C07282=1015.602,-60.319,395.785,165.379,57.389,160.207
C07283=1015.597,-60.568,395.794,165.376,57.396,160.208
C07284=1015.592,-60.819,395.805,165.373,57.403,160.208
C07285=1015.587,-61.068,395.815,165.370,57.410,160.209
C07286=1015.582,-61.318,395.825,165.367,57.417,160.210
C07287=1015.577,-61.568,395.835,165.364,57.424,160.210
C07288=1015.572,-61.818,395.845,165.361,57.431,160.211
C07289=1015.567,-62.067,395.855,165.358,57.438,160.211
C07290=1015.562,-62.317,395.865,165.356,57.444,160.212
C07291=1015.557,-62.567,395.875,165.353,57.451,160.212
C07292=1015.551,-62.817,395.885,165.351,57.458,160.213
C07293=1015.546,-63.066,395.895,165.348,57.465,160.213
C07294=1015.541,-63.316,395.905,165.345,57.472,160.214
C07295=1015.536,-63.566,395.915,165.342,57.479,160.215
C07296=1015.531,-63.816,395.925,165.339,57.486,160.215
C07297=1015.526,-64.065,395.935,165.337,57.493,160.216
C07298=1015.521,-64.315,395.945,165.334,57.500,160.216
C07299=1015.516,-64.565,395.955,165.331,57.507,160.217
C07300=1015.511,-64.814,395.964,165.328,57.514,160.217
C07301=1015.505,-65.064,395.975,165.325,57.521,160.218
C07302=1015.501,-65.314,395.984,165.322,57.528,160.218
C07303=1015.496,-65.563,395.994,165.320,57.534,160.219
C07304=1015.490,-65.813,396.004,165.317,57.541,160.219
C07305=1015.485,-66.063,396.014,165.314,57.548,160.220
C07306=1015.480,-66.313,396.024,165.311,57.555,160.220
C07307=1015.475,-66.562,396.034,165.308,57.562,160.221
C07308=1015.471,-66.812,396.043,165.306,57.568,160.222
C07309=1015.465,-67.062,396.053,165.303,57.575,160.222
C07310=1015.460,-67.312,396.063,165.300,57.582,160.223
C07311=1015.456,-67.561,396.073,165.297,57.589,160.223
C07312=1015.450,-67.811,396.083,165.295,57.595,160.224
C07313=1015.445,-68.061,396.093,165.292,57.602,160.224
C07314=1015.440,-68.310,396.103,165.289,57.609,160.225
C07315=1015.435,-68.561,396.112,165.286,57.616,160.225
C07316=1015.431,-68.811,396.123,165.284,57.622,160.226
C07317=1015.426,-69.060,396.132,165.281,57.629,160.226
C07318=1015.421,-69.323,396.142,165.278,57.636,160.227
C07319=1015.415,-69.600,396.154,165.274,57.644,160.227
C07320=1015.410,-69.877,396.164,165.272,57.651,160.228
C07321=1015.404,-70.154,396.176,165.269,57.659,160.229
C07322=1015.399,-70.432,396.186,165.266,57.667,160.229
C07323=1015.394,-70.682,396.196,165.263,57.673,160.230
C07324=1015.389,-70.931,396.206,165.260,57.680,160.230
C07325=1015.384,-71.182,396.215,165.257,57.687,160.231
C07326=1015.379,-71.431,396.225,165.255,57.692,160.231
C07327=1015.374,-71.681,396.235,165.252,57.700,160.232
C07328=1015.370,-71.930,396.245,165.249,57.707,160.232
C07329=1015.364,-72.181,396.254,165.246,57.713,160.232
C07330=1015.360,-72.430,396.264,165.244,57.719,160.233
C07331=1015.355,-72.680,396.274,165.241,57.726,160.234
C07332=1015.350,-72.930,396.283,165.237,57.733,160.234
C07333=1015.345,-73.180,396.293,165.236,57.739,160.235
C07334=1015.340,-73.429,396.303,165.232,57.746,160.235
C07335=1015.335,-73.678,396.313,165.229,57.753,160.235
C07336=1015.331,-73.928,396.322,165.227,57.759,160.236
C07337=1015.325,-74.179,396.332,165.224,57.766,160.236
C07338=1015.320,-74.428,396.342,165.221,57.773,160.237
C07339=1015.316,-74.678,396.351,165.219,57.779,160.237
C07340=1015.310,-74.927,396.360,165.216,57.786,160.238
C07341=1015.306,-75.177,396.369,165.213,57.793,160.238
C07342=1015.300,-75.427,396.379,165.210,57.800,160.239
C07343=1015.295,-75.677,396.388,165.207,57.806,160.239
C07344=1015.290,-75.926,396.397,165.205,57.813,160.240
C07345=1015.286,-76.176,396.407,165.202,57.820,160.240
C07346=1015.281,-76.426,396.416,165.199,57.827,160.241
C07347=1015.276,-76.676,396.425,165.196,57.833,160.241
C07348=1015.270,-76.926,396.434,165.194,57.840,160.242
C07349=1015.266,-77.176,396.444,165.191,57.847,160.243
C07350=1015.260,-77.425,396.453,165.187,57.853,160.243
C07351=1015.255,-77.675,396.462,165.185,57.860,160.243
C07352=1015.251,-77.925,396.471,165.182,57.867,160.244
C07353=1015.246,-78.175,396.480,165.180,57.874,160.245
C07354=1015.241,-78.424,396.490,165.176,57.880,160.245
C07355=1015.236,-78.675,396.499,165.174,57.887,160.246
C07356=1015.231,-78.924,396.509,165.171,57.893,160.246
C07357=1015.226,-79.174,396.517,165.168,57.900,160.246
C07358=1015.221,-79.424,396.526,165.166,57.907,160.247
C07359=1015.216,-79.673,396.536,165.163,57.913,160.247
C07360=1015.211,-79.923,396.545,165.160,57.920,160.248
C07361=1015.207,-80.173,396.554,165.158,57.927,160.249
///RCONF 1,0,0,0,1,0,0,0,0,0,0,0,0,0,0,0,0,0,0,0,0,0,0,0
C07362=1015.201,-80.423,396.564,165.155,57.933,160.249
C07363=1015.196,-80.673,396.572,165.152,57.940,160.249
C07364=1015.191,-80.923,396.582,165.149,57.947,160.250
C07365=1015.186,-81.173,396.590,165.146,57.954,160.250
C07366=1015.181,-81.423,396.599,165.144,57.960,160.251
C07367=1015.176,-81.672,396.608,165.141,57.967,160.251
C07368=1015.171,-81.921,396.617,165.138,57.974,160.252
C07369=1015.166,-82.171,396.626,165.135,57.981,160.252
C07370=1015.161,-82.421,396.634,165.131,57.988,160.253
C07371=1015.156,-82.671,396.643,165.130,57.994,160.253
C07372=1015.151,-82.921,396.652,165.127,58.001,160.254
C07373=1015.147,-83.171,396.661,165.123,58.008,160.254
C07374=1015.141,-83.421,396.670,165.120,58.015,160.255
C07375=1015.136,-83.670,396.679,165.119,58.021,160.255
C07376=1015.131,-83.920,396.688,165.115,58.028,160.256
C07377=1015.126,-84.169,396.696,165.112,58.035,160.256
C07378=1015.121,-84.419,396.705,165.109,58.042,160.257
C07379=1015.116,-84.669,396.714,165.107,58.048,160.257
C07380=1015.111,-84.919,396.722,165.104,58.055,160.258
C07381=1015.106,-85.169,396.731,165.101,58.062,160.258
C07382=1015.101,-85.419,396.740,165.098,58.068,160.258
C07383=1015.095,-85.698,396.750,165.096,58.076,160.259
C07384=1015.090,-85.978,396.760,165.093,58.083,160.260
C07385=1015.085,-86.257,396.769,165.089,58.090,160.260
C07386=1015.079,-86.536,396.779,165.086,58.098,160.261
C07387=1015.074,-86.786,396.788,165.083,58.105,160.261
C07388=1015.069,-87.036,396.797,165.081,58.111,160.262
C07389=1015.064,-87.285,396.806,165.078,58.118,160.262
C07390=1015.059,-87.535,396.815,165.074,58.124,160.262
C07391=1015.054,-87.785,396.823,165.073,58.131,160.263
C07392=1015.049,-88.035,396.832,165.069,58.137,160.263
C07393=1015.044,-88.285,396.841,165.066,58.144,160.264
C07394=1015.039,-88.535,396.849,165.064,58.150,160.264
C07395=1015.035,-88.784,396.858,165.061,58.157,160.265
C07396=1015.030,-89.034,396.866,165.058,58.163,160.265
C07397=1015.025,-89.283,396.875,165.056,58.170,160.266
C07398=1015.020,-89.534,396.883,165.053,58.176,160.266
C07399=1015.015,-89.784,396.892,165.050,58.183,160.266
C07400=1015.011,-90.034,396.901,165.047,58.189,160.267
C07401=1015.005,-90.284,396.909,165.044,58.196,160.267
C07402=1015.000,-90.533,396.918,165.042,58.202,160.268
C07403=1014.996,-90.783,396.926,165.039,58.209,160.268
C07404=1014.991,-91.032,396.935,165.036,58.216,160.269
C07405=1014.986,-91.282,396.944,165.033,58.222,160.269
C07406=1014.981,-91.532,396.952,165.031,58.229,160.270
C07407=1014.976,-91.782,396.961,165.028,58.235,160.270
C07408=1014.972,-92.032,396.969,165.025,58.241,160.270
C07409=1014.967,-92.281,396.977,165.023,58.248,160.271
C07410=1014.962,-92.531,396.987,165.020,58.254,160.271
C07411=1014.957,-92.781,396.995,165.016,58.260,160.271
C07412=1014.952,-93.031,397.003,165.014,58.267,160.272
C07413=1014.947,-93.281,397.013,165.011,58.273,160.272
C07414=1014.942,-93.531,397.021,165.009,58.279,160.273
C07415=1014.939,-93.781,397.029,165.005,58.286,160.273
C07416=1014.933,-94.030,397.038,165.003,58.292,160.274
C07417=1014.928,-94.280,397.046,165.000,58.299,160.274
C07418=1014.923,-94.530,397.055,164.998,58.305,160.274
C07419=1014.919,-94.779,397.063,164.995,58.312,160.275
C07420=1014.915,-95.030,397.072,164.992,58.318,160.275
C07421=1014.909,-95.279,397.080,164.989,58.324,160.276
C07422=1014.904,-95.529,397.089,164.987,58.330,160.276
C07423=1014.900,-95.778,397.097,164.983,58.336,160.276
C07424=1014.895,-96.029,397.105,164.981,58.343,160.277
C07425=1014.890,-96.278,397.114,164.978,58.349,160.277
C07426=1014.885,-96.528,397.123,164.976,58.355,160.278
C07427=1014.881,-96.777,397.131,164.972,58.362,160.278
C07428=1014.876,-97.028,397.139,164.970,58.368,160.278
C07429=1014.871,-97.278,397.148,164.968,58.374,160.279
C07430=1014.866,-97.528,397.156,164.965,58.381,160.279
C07431=1014.862,-97.777,397.165,164.962,58.387,160.280
C07432=1014.857,-98.027,397.173,164.959,58.393,160.280
C07433=1014.852,-98.277,397.181,164.957,58.399,160.280
C07434=1014.847,-98.527,397.188,164.953,58.405,160.281
C07435=1014.843,-98.777,397.198,164.951,58.412,160.281
C07436=1014.838,-99.027,397.205,164.948,58.418,160.282
C07437=1014.833,-99.276,397.213,164.945,58.425,160.282
C07438=1014.828,-99.526,397.221,164.943,58.431,160.282
C07439=1014.823,-99.776,397.230,164.939,58.438,160.283
C07440=1014.819,-100.026,397.237,164.937,58.444,160.283
C07441=1014.813,-100.275,397.246,164.934,58.450,160.283
C07442=1014.808,-100.526,397.253,164.932,58.457,160.284
C07443=1014.804,-100.775,397.261,164.929,58.463,160.284
C07444=1014.799,-101.025,397.269,164.926,58.469,160.285
C07445=1014.794,-101.275,397.278,164.923,58.475,160.285
C07446=1014.790,-101.525,397.286,164.920,58.481,160.285
C07447=1014.784,-101.806,397.295,164.918,58.488,160.286
C07448=1014.779,-102.088,397.304,164.915,58.496,160.286
C07449=1014.773,-102.369,397.313,164.911,58.503,160.287
C07450=1014.768,-102.651,397.322,164.908,58.510,160.287
C07451=1014.763,-102.900,397.330,164.906,58.516,160.288
C07452=1014.758,-103.150,397.338,164.902,58.523,160.288
C07453=1014.754,-103.399,397.346,164.900,58.529,160.288
C07454=1014.749,-103.650,397.354,164.897,58.535,160.289
C07455=1014.744,-103.900,397.361,164.894,58.541,160.289
C07456=1014.739,-104.149,397.370,164.892,58.547,160.289
C07457=1014.734,-104.399,397.377,164.889,58.554,160.290
C07458=1014.730,-104.649,397.385,164.887,58.560,160.290
C07459=1014.725,-104.899,397.393,164.883,58.566,160.291
C07460=1014.720,-105.148,397.401,164.881,58.572,160.291
C07461=1014.715,-105.399,397.408,164.879,58.578,160.291
C07462=1014.711,-105.648,397.417,164.875,58.585,160.292
C07463=1014.706,-105.898,397.425,164.873,58.590,160.292
C07464=1014.702,-106.148,397.432,164.870,58.597,160.292
C07465=1014.697,-106.398,397.441,164.867,58.603,160.293
C07466=1014.692,-106.648,397.449,164.865,58.609,160.293
C07467=1014.688,-106.898,397.456,164.862,58.615,160.293
C07468=1014.683,-107.148,397.464,164.859,58.621,160.294
C07469=1014.678,-107.397,397.472,164.856,58.627,160.294
C07470=1014.673,-107.647,397.480,164.853,58.633,160.294
C07471=1014.669,-107.897,397.487,164.851,58.639,160.295
C07472=1014.664,-108.147,397.495,164.848,58.646,160.295
C07473=1014.659,-108.396,397.503,164.845,58.652,160.296
C07474=1014.654,-108.646,397.510,164.843,58.658,160.296
C07475=1014.649,-108.896,397.518,164.840,58.664,160.296
C07476=1014.645,-109.146,397.525,164.837,58.670,160.297
C07477=1014.640,-109.396,397.533,164.834,58.676,160.297
C07478=1014.635,-109.646,397.540,164.832,58.682,160.297
C07479=1014.630,-109.896,397.548,164.829,58.688,160.298
C07480=1014.626,-110.145,397.555,164.826,58.695,160.298
C07481=1014.621,-110.395,397.564,164.824,58.701,160.298
C07482=1014.616,-110.645,397.571,164.821,58.707,160.299
C07483=1014.611,-110.894,397.578,164.818,58.713,160.299
C07484=1014.606,-111.144,397.586,164.816,58.719,160.299
C07485=1014.602,-111.394,397.593,164.812,58.725,160.300
C07486=1014.597,-111.644,397.601,164.810,58.731,160.300
C07487=1014.593,-111.894,397.608,164.808,58.737,160.300
C07488=1014.588,-112.144,397.616,164.805,58.743,160.301
C07489=1014.583,-112.394,397.623,164.802,58.750,160.301
C07490=1014.579,-112.644,397.631,164.800,58.756,160.302
C07491=1014.573,-112.894,397.638,164.797,58.762,160.302
C07492=1014.569,-113.143,397.645,164.794,58.768,160.302
C07493=1014.564,-113.393,397.653,164.791,58.774,160.303
C07494=1014.560,-113.643,397.661,164.789,58.779,160.303
C07495=1014.555,-113.893,397.668,164.786,58.785,160.303
C07496=1014.551,-114.143,397.675,164.783,58.792,160.303
C07497=1014.546,-114.393,397.683,164.781,58.798,160.304
C07498=1014.541,-114.643,397.691,164.778,58.804,160.304
C07499=1014.536,-114.892,397.697,164.776,58.810,160.305
C07500=1014.531,-115.142,397.705,164.772,58.815,160.305
C07501=1014.527,-115.392,397.713,164.770,58.821,160.305
C07502=1014.523,-115.641,397.720,164.767,58.827,160.305
C07503=1014.517,-115.891,397.727,164.764,58.834,160.306
C07504=1014.513,-116.141,397.735,164.762,58.840,160.306
C07505=1014.508,-116.391,397.742,164.759,58.845,160.306
C07506=1014.504,-116.642,397.749,164.757,58.851,160.307
C07507=1014.499,-116.891,397.756,164.753,58.857,160.307
C07508=1014.494,-117.141,397.763,164.751,58.863,160.307
C07509=1014.490,-117.390,397.771,164.748,58.869,160.308
C07510=1014.485,-117.641,397.778,164.746,58.875,160.308
C07511=1014.480,-117.922,397.786,164.743,58.881,160.308
C07512=1014.474,-118.204,397.794,164.739,58.888,160.308
C07513=1014.469,-118.485,397.802,164.737,58.895,160.309
C07514=1014.464,-118.767,397.811,164.733,58.901,160.309
C07515=1014.460,-119.017,397.817,164.731,58.907,160.310
C07516=1014.455,-119.266,397.824,164.729,58.913,160.310
C07517=1014.450,-119.517,397.832,164.726,58.919,160.310
C07518=1014.445,-119.766,397.839,164.723,58.925,160.311
C07519=1014.441,-120.016,397.846,164.720,58.931,160.311
C07520=1014.436,-120.266,397.853,164.718,58.937,160.311
C07521=1014.431,-120.516,397.861,164.715,58.942,160.311
C07522=1014.427,-120.766,397.868,164.712,58.948,160.312
C07523=1014.422,-121.016,397.874,164.710,58.954,160.312
C07524=1014.418,-121.265,397.881,164.707,58.959,160.312
C07525=1014.413,-121.515,397.889,164.704,58.966,160.313
C07526=1014.408,-121.766,397.895,164.702,58.972,160.313
C07527=1014.403,-122.015,397.903,164.699,58.977,160.313
C07528=1014.399,-122.265,397.910,164.696,58.983,160.313
C07529=1014.394,-122.515,397.916,164.694,58.989,160.314
C07530=1014.390,-122.764,397.924,164.691,58.994,160.314
C07531=1014.386,-123.014,397.931,164.689,59.000,160.314
C07532=1014.380,-123.265,397.937,164.686,59.006,160.315
C07533=1014.376,-123.514,397.945,164.684,59.012,160.315
C07534=1014.372,-123.765,397.952,164.680,59.018,160.315
C07535=1014.367,-124.014,397.958,164.677,59.023,160.315
C07536=1014.362,-124.264,397.966,164.675,59.029,160.316
C07537=1014.358,-124.514,397.972,164.672,59.034,160.316
C07538=1014.353,-124.763,397.979,164.670,59.040,160.316
C07539=1014.349,-125.013,397.986,164.667,59.046,160.316
C07540=1014.343,-125.263,397.993,164.665,59.052,160.317
C07541=1014.339,-125.514,398.000,164.662,59.058,160.317
C07542=1014.334,-125.763,398.007,164.659,59.063,160.317
C07543=1014.330,-126.013,398.013,164.657,59.069,160.318
C07544=1014.325,-126.263,398.020,164.654,59.074,160.318
C07545=1014.321,-126.513,398.027,164.652,59.080,160.318
C07546=1014.316,-126.762,398.034,164.650,59.086,160.319
C07547=1014.312,-127.012,398.040,164.647,59.091,160.319
C07548=1014.307,-127.262,398.047,164.643,59.098,160.319
C07549=1014.303,-127.512,398.054,164.641,59.103,160.319
C07550=1014.298,-127.761,398.061,164.638,59.109,160.320
C07551=1014.294,-128.012,398.067,164.635,59.114,160.320
C07552=1014.289,-128.261,398.074,164.633,59.120,160.320
C07553=1014.284,-128.511,398.082,164.631,59.125,160.320
C07554=1014.281,-128.760,398.090,164.628,59.130,160.320
C07555=1014.277,-129.009,398.098,164.625,59.134,160.320
C07556=1014.274,-129.259,398.107,164.623,59.136,160.320
C07557=1014.272,-129.509,398.117,164.620,59.140,160.320
C07558=1014.269,-129.759,398.127,164.618,59.143,160.320
C07559=1014.266,-130.008,398.138,164.617,59.144,160.320
C07560=1014.265,-130.258,398.149,164.613,59.146,160.319
C07561=1014.264,-130.507,398.162,164.611,59.146,160.318
C07562=1014.263,-130.757,398.174,164.609,59.147,160.318
C07563=1014.262,-131.006,398.188,164.607,59.147,160.317
C07564=1014.262,-131.256,398.202,164.605,59.146,160.317
C07565=1014.261,-131.506,398.216,164.602,59.145,160.316
C07566=1014.262,-131.755,398.231,164.601,59.143,160.315
C07567=1014.263,-132.005,398.247,164.599,59.141,160.314
C07568=1014.264,-132.255,398.263,164.597,59.138,160.313
C07569=1014.264,-132.505,398.281,164.594,59.135,160.311
C07570=1014.267,-132.754,398.298,164.593,59.132,160.310
C07571=1014.269,-133.004,398.316,164.591,59.128,160.309
C07572=1014.271,-133.254,398.335,164.589,59.122,160.307
C07573=1014.274,-133.504,398.354,164.587,59.117,160.306
C07574=1014.277,-133.753,398.374,164.585,59.111,160.304
C07575=1014.043,-133.779,397.962,164.561,59.455,160.360
C07576=1014.040,-133.530,397.942,164.563,59.460,160.362
C07577=1014.036,-133.281,397.922,164.565,59.466,160.363
C07578=1014.035,-133.031,397.904,164.567,59.470,160.365
C07579=1014.032,-132.780,397.885,164.569,59.474,160.366
C07580=1014.031,-132.531,397.868,164.571,59.478,160.368
C07581=1014.029,-132.282,397.851,164.573,59.482,160.369
C07582=1014.028,-132.032,397.834,164.575,59.484,160.370
C07583=1014.028,-131.782,397.819,164.576,59.486,160.371
C07584=1014.027,-131.533,397.804,164.579,59.488,160.372
C07585=1014.027,-131.283,397.789,164.580,59.489,160.372
C07586=1014.027,-131.033,397.775,164.583,59.490,160.373
C07587=1014.028,-130.783,397.762,164.585,59.490,160.374
C07588=1014.029,-130.534,397.749,164.588,59.490,160.375
C07589=1014.030,-130.284,397.736,164.590,59.489,160.375
C07590=1014.032,-130.035,397.725,164.592,59.487,160.375
C07591=1014.034,-129.785,397.714,164.595,59.485,160.376
C07592=1014.037,-129.535,397.704,164.596,59.483,160.376
C07593=1014.039,-129.285,397.694,164.599,59.480,160.376
C07594=1014.043,-129.036,397.685,164.601,59.477,160.376
C07595=1014.046,-128.786,397.676,164.604,59.473,160.376
C07596=1014.050,-128.536,397.668,164.607,59.469,160.377
C07597=1014.054,-128.287,397.661,164.609,59.464,160.376
C07598=1014.059,-128.037,397.655,164.612,59.459,160.376
C07599=1014.063,-127.788,397.647,164.614,59.453,160.376
C07600=1014.068,-127.539,397.641,164.617,59.447,160.376
C07601=1014.072,-127.288,397.634,164.620,59.442,160.375
C07602=1014.077,-127.038,397.628,164.622,59.436,160.375
C07603=1014.081,-126.789,397.620,164.625,59.431,160.375
C07604=1014.086,-126.539,397.614,164.628,59.425,160.375
C07605=1014.090,-126.289,397.607,164.629,59.420,160.374
C07606=1014.095,-126.039,397.601,164.632,59.415,160.374
C07607=1014.100,-125.790,397.593,164.634,59.409,160.373
C07608=1014.104,-125.540,397.587,164.637,59.403,160.373
C07609=1014.108,-125.289,397.581,164.639,59.397,160.373
C07610=1014.113,-125.040,397.574,164.642,59.392,160.373
C07611=1014.118,-124.790,397.567,164.645,59.387,160.373
C07612=1014.123,-124.540,397.560,164.647,59.381,160.372
C07613=1014.127,-124.289,397.553,164.650,59.375,160.372
C07614=1014.132,-124.040,397.546,164.652,59.369,160.372
C07615=1014.137,-123.791,397.539,164.655,59.364,160.372
C07616=1014.141,-123.540,397.532,164.658,59.359,160.371
C07617=1014.145,-123.291,397.525,164.660,59.353,160.371
C07618=1014.150,-123.041,397.519,164.663,59.348,160.371
C07619=1014.154,-122.791,397.511,164.665,59.342,160.370
C07620=1014.159,-122.541,397.504,164.668,59.336,160.370
C07621=1014.164,-122.291,397.498,164.670,59.330,160.370
C07622=1014.168,-122.041,397.490,164.673,59.325,160.370
C07623=1014.172,-121.791,397.484,164.676,59.319,160.369
C07624=1014.178,-121.542,397.477,164.678,59.314,160.369
C07625=1014.182,-121.292,397.469,164.681,59.308,160.369
C07626=1014.186,-121.042,397.463,164.685,59.302,160.369
C07627=1014.191,-120.792,397.456,164.687,59.296,160.368
C07628=1014.196,-120.542,397.448,164.690,59.291,160.368
C07629=1014.200,-120.292,397.441,164.692,59.285,160.368
C07630=1014.205,-120.042,397.435,164.695,59.280,160.368
C07631=1014.210,-119.793,397.427,164.697,59.274,160.367
C07632=1014.214,-119.543,397.420,164.699,59.268,160.367
C07633=1014.219,-119.292,397.413,164.702,59.262,160.367
C07634=1014.224,-119.043,397.406,164.705,59.256,160.366
C07635=1014.228,-118.793,397.398,164.707,59.251,160.366
C07636=1014.233,-118.512,397.391,164.710,59.244,160.366
C07637=1014.239,-118.230,397.383,164.713,59.237,160.365
C07638=1014.244,-117.949,397.375,164.717,59.231,160.365
C07639=1014.249,-117.668,397.367,164.719,59.225,160.365
C07640=1014.254,-117.418,397.359,164.722,59.218,160.365
C07641=1014.258,-117.167,397.352,164.725,59.212,160.364
C07642=1014.263,-116.918,397.345,164.728,59.207,160.364
C07643=1014.267,-116.668,397.338,164.730,59.201,160.364
C07644=1014.272,-116.418,397.330,164.732,59.195,160.363
C07645=1014.276,-116.168,397.323,164.735,59.190,160.363
C07646=1014.281,-115.918,397.317,164.738,59.183,160.363
C07647=1014.286,-115.668,397.309,164.741,59.177,160.362
C07648=1014.291,-115.419,397.302,164.743,59.172,160.362
C07649=1014.295,-115.169,397.294,164.746,59.166,160.362
C07650=1014.300,-114.920,397.287,164.748,59.160,160.361
C07651=1014.305,-114.669,397.280,164.751,59.154,160.361
C07652=1014.309,-114.420,397.272,164.754,59.149,160.361
C07653=1014.314,-114.170,397.265,164.756,59.143,160.361
C07654=1014.319,-113.920,397.257,164.759,59.137,160.360
C07655=1014.323,-113.670,397.250,164.762,59.131,160.360
C07656=1014.327,-113.420,397.242,164.764,59.125,160.360
C07657=1014.333,-113.170,397.235,164.767,59.119,160.359
C07658=1014.337,-112.921,397.228,164.769,59.113,160.359
C07659=1014.342,-112.671,397.220,164.772,59.108,160.359
C07660=1014.346,-112.420,397.213,164.775,59.102,160.358
C07661=1014.351,-112.171,397.205,164.778,59.095,160.358
C07662=1014.355,-111.921,397.198,164.780,59.089,160.358
C07663=1014.360,-111.671,397.190,164.782,59.083,160.357
C07664=1014.365,-111.422,397.182,164.785,59.078,160.357
C07665=1014.370,-111.172,397.176,164.789,59.072,160.357
C07666=1014.375,-110.922,397.168,164.791,59.066,160.356
C07667=1014.379,-110.672,397.160,164.793,59.060,160.356
C07668=1014.384,-110.422,397.153,164.795,59.054,160.356
C07669=1014.388,-110.172,397.145,164.799,59.047,160.355
C07670=1014.393,-109.923,397.138,164.802,59.042,160.355
C07671=1014.398,-109.672,397.130,164.804,59.036,160.355
C07672=1014.402,-109.423,397.123,164.807,59.029,160.355
C07673=1014.407,-109.172,397.115,164.810,59.024,160.354
C07674=1014.412,-108.923,397.108,164.812,59.018,160.354
C07675=1014.417,-108.673,397.101,164.815,59.011,160.353
C07676=1014.421,-108.423,397.093,164.818,59.005,160.353
C07677=1014.426,-108.174,397.085,164.820,58.999,160.353
C07678=1014.431,-107.924,397.077,164.823,58.993,160.352
C07679=1014.435,-107.674,397.070,164.825,58.987,160.352
C07680=1014.440,-107.424,397.062,164.828,58.981,160.351
C07681=1014.445,-107.174,397.054,164.831,58.974,160.351
C07682=1014.450,-106.924,397.047,164.833,58.968,160.351
C07683=1014.454,-106.675,397.039,164.836,58.963,160.351
C07684=1014.459,-106.424,397.031,164.840,58.957,160.350
C07685=1014.464,-106.175,397.023,164.842,58.951,160.350
C07686=1014.469,-105.924,397.016,164.844,58.945,160.350
C07687=1014.473,-105.675,397.008,164.848,58.938,160.349
C07688=1014.478,-105.425,397.000,164.850,58.932,160.349
C07689=1014.483,-105.175,396.992,164.852,58.926,160.348
C07690=1014.488,-104.926,396.984,164.855,58.920,160.348
C07691=1014.492,-104.676,396.976,164.858,58.914,160.348
C07692=1014.496,-104.425,396.968,164.860,58.908,160.347
C07693=1014.501,-104.176,396.960,164.863,58.902,160.347
C07694=1014.506,-103.926,396.952,164.866,58.896,160.347
C07695=1014.510,-103.676,396.945,164.868,58.890,160.346
C07696=1014.516,-103.427,396.936,164.871,58.883,160.346
C07697=1014.520,-103.177,396.929,164.874,58.877,160.346
C07698=1014.525,-102.927,396.921,164.877,58.871,160.345
C07699=1014.530,-102.678,396.913,164.879,58.865,160.345
C07700=1014.535,-102.396,396.904,164.882,58.858,160.344
C07701=1014.540,-102.115,396.895,164.885,58.850,160.344
C07702=1014.545,-101.833,396.886,164.888,58.844,160.344
C07703=1014.551,-101.552,396.877,164.891,58.837,160.343
C07704=1014.556,-101.302,396.869,164.894,58.830,160.343
C07705=1014.561,-101.053,396.861,164.896,58.825,160.342
C07706=1014.566,-100.803,396.853,164.900,58.818,160.342
C07707=1014.570,-100.554,396.845,164.902,58.812,160.342
C07708=1014.575,-100.303,396.838,164.905,58.805,160.341
C07709=1014.580,-100.053,396.830,164.907,58.799,160.341
C07710=1014.584,-99.804,396.821,164.911,58.793,160.341
C07711=1014.589,-99.553,396.813,164.913,58.787,160.340
C07712=1014.594,-99.304,396.805,164.916,58.780,160.340
C07713=1014.599,-99.054,396.797,164.918,58.774,160.339
C07714=1014.604,-98.804,396.789,164.921,58.767,160.339
C07715=1014.608,-98.555,396.782,164.924,58.761,160.338
C07716=1014.614,-98.305,396.773,164.927,58.755,160.338
C07717=1014.619,-98.054,396.765,164.929,58.749,160.338
C07718=1014.622,-97.805,396.757,164.932,58.742,160.337
C07719=1014.628,-97.555,396.748,164.934,58.736,160.337
C07720=1014.633,-97.305,396.740,164.937,58.730,160.336
C07721=1014.637,-97.055,396.731,164.940,58.723,160.336
C07722=1014.642,-96.806,396.723,164.942,58.717,160.336
C07723=1014.646,-96.555,396.715,164.946,58.711,160.335
C07724=1014.651,-96.306,396.706,164.948,58.705,160.335
C07725=1014.656,-96.057,396.698,164.951,58.699,160.335
C07726=1014.660,-95.806,396.690,164.954,58.693,160.334
C07727=1014.665,-95.556,396.681,164.956,58.687,160.334
C07728=1014.669,-95.307,396.673,164.959,58.680,160.334
C07729=1014.675,-95.057,396.664,164.961,58.674,160.333
C07730=1014.680,-94.807,396.656,164.964,58.667,160.333
C07731=1014.684,-94.557,396.647,164.967,58.661,160.332
C07732=1014.689,-94.308,396.639,164.970,58.655,160.332
C07733=1014.694,-94.058,396.631,164.972,58.649,160.332
C07734=1014.698,-93.808,396.622,164.975,58.642,160.331
C07735=1014.704,-93.558,396.614,164.977,58.636,160.331
C07736=1014.707,-93.309,396.605,164.981,58.629,160.330
C07737=1014.713,-93.059,396.597,164.983,58.624,160.330
C07738=1014.718,-92.808,396.589,164.987,58.617,160.330
C07739=1014.722,-92.558,396.580,164.988,58.610,160.329
C07740=1014.727,-92.309,396.572,164.992,58.604,160.329
C07741=1014.731,-92.059,396.563,164.994,58.598,160.328
C07742=1014.737,-91.810,396.554,164.997,58.591,160.328
C07743=1014.742,-91.560,396.546,165.000,58.585,160.327
C07744=1014.746,-91.309,396.537,165.002,58.579,160.327
C07745=1014.751,-91.060,396.529,165.006,58.572,160.327
C07746=1014.755,-90.810,396.520,165.008,58.566,160.326
C07747=1014.761,-90.561,396.512,165.011,58.559,160.326
C07748=1014.766,-90.311,396.503,165.013,58.553,160.325
C07749=1014.770,-90.061,396.494,165.016,58.546,160.325
C07750=1014.776,-89.811,396.486,165.019,58.540,160.325
C07751=1014.779,-89.561,396.478,165.021,58.533,160.324
C07752=1014.785,-89.311,396.469,165.025,58.527,160.324
C07753=1014.790,-89.062,396.461,165.027,58.521,160.323
C07754=1014.794,-88.812,396.451,165.030,58.514,160.323
C07755=1014.800,-88.562,396.443,165.033,58.507,160.322
C07756=1014.804,-88.312,396.434,165.035,58.501,160.322
C07757=1014.809,-88.062,396.425,165.038,58.494,160.321
C07758=1014.814,-87.813,396.417,165.041,58.487,160.321
C07759=1014.819,-87.563,396.408,165.043,58.481,160.320
C07760=1014.824,-87.313,396.400,165.046,58.474,160.320
C07761=1014.828,-87.063,396.391,165.049,58.468,160.320
C07762=1014.834,-86.814,396.382,165.051,58.461,160.319
C07763=1014.839,-86.564,396.374,165.055,58.455,160.319
C07764=1014.844,-86.284,396.364,165.057,58.447,160.318
C07765=1014.850,-86.006,396.354,165.061,58.440,160.318
C07766=1014.855,-85.726,396.344,165.063,58.432,160.317
C07767=1014.860,-85.447,396.335,165.066,58.425,160.316
C07768=1014.865,-85.197,396.327,165.070,58.419,160.316
C07769=1014.870,-84.947,396.318,165.072,58.411,160.316
C07770=1014.875,-84.697,396.309,165.074,58.405,160.315
C07771=1014.880,-84.448,396.299,165.078,58.398,160.315
C07772=1014.885,-84.198,396.291,165.080,58.391,160.314
C07773=1014.891,-83.948,396.282,165.084,58.385,160.314
C07774=1014.895,-83.698,396.273,165.085,58.378,160.313
C07775=1014.900,-83.449,396.265,165.088,58.371,160.312
C07776=1014.905,-83.199,396.256,165.092,58.365,160.312
C07777=1014.910,-82.949,396.247,165.094,58.358,160.312
C07778=1014.915,-82.699,396.238,165.096,58.351,160.311
C07779=1014.920,-82.449,396.230,165.100,58.345,160.311
C07780=1014.925,-82.200,396.221,165.102,58.338,160.310
C07781=1014.930,-81.950,396.212,165.105,58.330,160.310
C07782=1014.935,-81.700,396.204,165.109,58.324,160.309
C07783=1014.939,-81.450,396.195,165.110,58.317,160.309
C07784=1014.945,-81.201,396.185,165.113,58.310,160.308
C07785=1014.950,-80.951,396.176,165.116,58.303,160.308
C07786=1014.955,-80.701,396.168,165.119,58.297,160.307
C07787=1014.960,-80.451,396.159,165.122,58.290,160.307
C07788=1014.965,-80.201,396.150,165.124,58.283,160.306
C07789=1014.969,-79.951,396.141,165.127,58.277,160.306
C07790=1014.974,-79.702,396.131,165.130,58.270,160.305
C07791=1014.980,-79.451,396.122,165.133,58.264,160.305
C07792=1014.984,-79.201,396.113,165.135,58.257,160.304
C07793=1014.989,-78.952,396.104,165.138,58.250,160.304
C07794=1014.994,-78.702,396.095,165.141,58.244,160.303
///RCONF 1,0,0,0,0,0,0,0,0,0,0,0,0,0,0,0,0,0,0,0,0,0,0,0
C07795=1014.999,-78.452,396.086,165.143,58.237,160.303
C07796=1015.004,-78.203,396.076,165.147,58.230,160.302
C07797=1015.009,-77.953,396.068,165.150,58.223,160.302
C07798=1015.014,-77.703,396.059,165.151,58.217,160.301
C07799=1015.018,-77.454,396.049,165.155,58.210,160.301
C07800=1015.023,-77.204,396.040,165.158,58.203,160.300
C07801=1015.029,-76.954,396.031,165.160,58.196,160.300
C07802=1015.034,-76.704,396.021,165.163,58.190,160.299
C07803=1015.038,-76.454,396.012,165.166,58.183,160.299
C07804=1015.044,-76.205,396.003,165.168,58.176,160.298
C07805=1015.048,-75.955,395.994,165.171,58.169,160.298
C07806=1015.053,-75.705,395.984,165.174,58.163,160.297
C07807=1015.058,-75.455,395.976,165.176,58.156,160.297
C07808=1015.063,-75.205,395.966,165.179,58.149,160.296
C07809=1015.068,-74.955,395.956,165.182,58.142,160.296
C07810=1015.073,-74.705,395.947,165.186,58.135,160.295
C07811=1015.078,-74.456,395.938,165.187,58.129,160.295
C07812=1015.083,-74.206,395.929,165.190,58.122,160.294
C07813=1015.087,-73.956,395.919,165.194,58.115,160.294
C07814=1015.092,-73.707,395.909,165.195,58.109,160.293
C07815=1015.097,-73.456,395.899,165.199,58.102,160.293
C07816=1015.102,-73.207,395.889,165.202,58.095,160.292
C07817=1015.107,-72.958,395.880,165.204,58.089,160.292
C07818=1015.111,-72.707,395.871,165.207,58.082,160.291
C07819=1015.116,-72.458,395.861,165.210,58.075,160.291
C07820=1015.121,-72.208,395.851,165.212,58.069,160.290
C07821=1015.126,-71.958,395.842,165.215,58.062,160.290
C07822=1015.131,-71.709,395.832,165.218,58.055,160.289
C07823=1015.136,-71.459,395.822,165.221,58.049,160.289
C07824=1015.141,-71.208,395.813,165.223,58.042,160.288
C07825=1015.146,-70.959,395.803,165.226,58.035,160.288
C07826=1015.150,-70.710,395.793,165.229,58.029,160.288
C07827=1015.155,-70.460,395.783,165.231,58.022,160.287
C07828=1015.161,-70.182,395.772,165.235,58.015,160.286
C07829=1015.167,-69.906,395.763,165.237,58.007,160.286
C07830=1015.172,-69.628,395.751,165.241,57.999,160.285
C07831=1015.178,-69.350,395.741,165.244,57.992,160.285
C07832=1015.183,-69.101,395.731,165.247,57.985,160.284
C07833=1015.188,-68.852,395.721,165.249,57.979,160.283
C07834=1015.192,-68.602,395.711,165.251,57.972,160.283
C07835=1015.197,-68.351,395.702,165.255,57.965,160.283
C07836=1015.202,-68.102,395.692,165.258,57.958,160.282
C07837=1015.207,-67.853,395.682,165.261,57.951,160.282
C07838=1015.213,-67.603,395.672,165.262,57.944,160.281
C07839=1015.217,-67.353,395.662,165.265,57.937,160.280
C07840=1015.221,-67.103,395.653,165.268,57.930,160.280
C07841=1015.227,-66.853,395.642,165.272,57.924,160.279
C07842=1015.231,-66.603,395.633,165.274,57.917,160.279
C07843=1015.236,-66.354,395.623,165.276,57.910,160.278
C07844=1015.242,-66.104,395.613,165.279,57.903,160.278
C07845=1015.247,-65.854,395.603,165.282,57.896,160.277
C07846=1015.251,-65.604,395.594,165.285,57.889,160.276
C07847=1015.257,-65.354,395.584,165.288,57.882,160.276
C07848=1015.261,-65.105,395.574,165.291,57.876,160.276
C07849=1015.266,-64.855,395.564,165.293,57.869,160.275
C07850=1015.272,-64.605,395.554,165.296,57.862,160.274
C07851=1015.276,-64.356,395.544,165.299,57.855,160.274
C07852=1015.282,-64.106,395.534,165.301,57.848,160.273
C07853=1015.287,-63.856,395.524,165.304,57.841,160.273
C07854=1015.292,-63.607,395.514,165.307,57.834,160.272
C07855=1015.297,-63.357,395.504,165.310,57.827,160.272
C07856=1015.302,-63.107,395.495,165.312,57.820,160.271
C07857=1015.307,-62.857,395.485,165.315,57.813,160.270
C07858=1015.312,-62.607,395.475,165.318,57.806,160.270
C07859=1015.317,-62.358,395.465,165.321,57.799,160.269
C07860=1015.322,-62.108,395.455,165.323,57.792,160.269
C07861=1015.327,-61.858,395.445,165.326,57.785,160.268
C07862=1015.332,-61.608,395.435,165.329,57.778,160.268
C07863=1015.337,-61.359,395.425,165.332,57.771,160.267
C07864=1015.343,-61.109,395.415,165.335,57.764,160.267
C07865=1015.347,-60.859,395.405,165.338,57.757,160.266
C07866=1015.352,-60.610,395.396,165.339,57.750,160.265
C07867=1015.358,-60.360,395.386,165.342,57.743,160.264
C07868=1015.363,-60.110,395.376,165.345,57.736,160.264
C07869=1015.368,-59.860,395.366,165.348,57.729,160.263
C07870=1015.372,-59.611,395.355,165.351,57.722,160.263
C07871=1015.377,-59.360,395.345,165.353,57.715,160.262
C07872=1015.382,-59.111,395.335,165.356,57.707,160.262
C07873=1015.388,-58.861,395.325,165.359,57.700,160.261
C07874=1015.393,-58.612,395.315,165.361,57.693,160.260
C07875=1015.398,-58.361,395.305,165.364,57.686,160.260
C07876=1015.403,-58.144,395.296,165.367,57.680,160.259
C07877=1015.407,-57.927,395.287,165.369,57.674,160.259
C07878=1015.412,-57.710,395.279,165.372,57.667,160.258
C07879=1015.416,-57.492,395.270,165.374,57.661,160.258
C07880=1015.420,-57.274,395.261,165.376,57.654,160.257
C07881=1015.425,-57.057,395.252,165.379,57.649,160.257
C07882=1015.430,-56.839,395.243,165.382,57.642,160.256
C07883=1015.434,-56.622,395.235,165.384,57.636,160.256
C07884=1015.440,-56.372,395.225,165.387,57.629,160.255
C07885=1015.444,-56.123,395.215,165.390,57.622,160.255
C07886=1015.449,-55.873,395.204,165.392,57.614,160.254
C07887=1015.455,-55.623,395.194,165.395,57.607,160.253
C07888=1015.460,-55.374,395.184,165.398,57.600,160.253
C07889=1015.465,-55.124,395.174,165.400,57.592,160.252
C07890=1015.470,-54.874,395.164,165.403,57.585,160.251
C07891=1015.475,-54.624,395.154,165.406,57.578,160.251
C07892=1015.483,-54.283,395.140,165.409,57.568,160.250
C07893=1015.490,-53.943,395.126,165.413,57.559,160.249
C07894=1015.497,-53.601,395.112,165.418,57.548,160.248
C07895=1015.504,-53.261,395.099,165.421,57.538,160.247
C07896=1015.509,-53.012,395.088,165.424,57.531,160.247
C07897=1015.515,-52.762,395.078,165.426,57.523,160.246
C07898=1015.520,-52.512,395.068,165.429,57.516,160.245
C07899=1015.525,-52.262,395.058,165.432,57.509,160.245
C07900=1015.530,-52.012,395.047,165.434,57.502,160.244
C07901=1015.535,-51.763,395.036,165.437,57.495,160.243
C07902=1015.540,-51.513,395.026,165.441,57.486,160.243
C07903=1015.546,-51.263,395.016,165.443,57.479,160.242
C07904=1015.551,-51.014,395.006,165.446,57.472,160.241
C07905=1015.556,-50.764,394.995,165.448,57.466,160.241
C07906=1015.561,-50.513,394.985,165.451,57.458,160.240
C07907=1015.566,-50.264,394.973,165.453,57.451,160.239
C07908=1015.571,-50.014,394.963,165.456,57.444,160.239
C07909=1015.576,-49.764,394.952,165.459,57.437,160.238
C07910=1015.581,-49.514,394.942,165.462,57.430,160.238
C07911=1015.586,-49.266,394.931,165.465,57.423,160.237
C07912=1015.591,-49.015,394.920,165.468,57.415,160.236
C07913=1015.597,-48.766,394.910,165.470,57.408,160.236
C07914=1015.601,-48.516,394.899,165.473,57.401,160.235
C07915=1015.607,-48.266,394.888,165.476,57.394,160.235
C07916=1015.611,-48.016,394.878,165.479,57.387,160.234
C07917=1015.617,-47.767,394.867,165.482,57.380,160.233
C07918=1015.622,-47.517,394.856,165.483,57.373,160.232
C07919=1015.627,-47.267,394.845,165.486,57.366,160.232
C07920=1015.632,-47.018,394.834,165.489,57.359,160.231
C07921=1015.637,-46.767,394.824,165.492,57.351,160.231
C07922=1015.642,-46.518,394.813,165.495,57.344,160.230
C07923=1015.648,-46.269,394.802,165.498,57.337,160.229
C07924=1015.652,-46.018,394.791,165.500,57.330,160.229
C07925=1015.658,-45.769,394.780,165.503,57.323,160.228
C07926=1015.662,-45.519,394.770,165.506,57.316,160.228
C07927=1015.668,-45.270,394.759,165.508,57.308,160.227
C07928=1015.673,-45.020,394.747,165.511,57.301,160.226
C07929=1015.678,-44.770,394.737,165.514,57.294,160.226
C07930=1015.683,-44.521,394.727,165.516,57.286,160.225
C07931=1015.688,-44.271,394.715,165.519,57.279,160.224
C07932=1015.694,-44.021,394.705,165.522,57.272,160.224
C07933=1015.699,-43.771,394.694,165.525,57.265,160.223
C07934=1015.705,-43.522,394.683,165.528,57.258,160.222
C07935=1015.709,-43.272,394.672,165.530,57.251,160.222
C07936=1015.714,-43.023,394.662,165.533,57.243,160.221
C07937=1015.719,-42.773,394.650,165.536,57.236,160.220
C07938=1015.725,-42.523,394.640,165.538,57.228,160.220
C07939=1015.730,-42.273,394.628,165.541,57.221,160.219
C07940=1015.736,-42.023,394.618,165.544,57.214,160.218
C07941=1015.740,-41.774,394.607,165.546,57.207,160.218
C07942=1015.745,-41.524,394.596,165.549,57.199,160.217
C07943=1015.750,-41.274,394.585,165.553,57.192,160.216
C07944=1015.756,-41.025,394.574,165.555,57.184,160.216
C07945=1015.761,-40.774,394.563,165.558,57.177,160.215
C07946=1015.767,-40.525,394.552,165.561,57.169,160.214
C07947=1015.772,-40.275,394.541,165.564,57.162,160.214
C07948=1015.777,-40.026,394.530,165.566,57.155,160.213
C07949=1015.781,-39.776,394.520,165.569,57.148,160.212
C07950=1015.787,-39.527,394.509,165.571,57.140,160.211
C07951=1015.792,-39.277,394.497,165.574,57.133,160.211
C07952=1015.797,-39.027,394.486,165.577,57.126,160.210
C07953=1015.803,-38.777,394.475,165.580,57.118,160.209
C07954=1015.808,-38.528,394.463,165.583,57.111,160.209
C07955=1015.813,-38.278,394.452,165.586,57.104,160.208
C07956=1015.818,-38.002,394.440,165.588,57.097,160.208
C07957=1015.824,-37.726,394.427,165.591,57.089,160.207
C07958=1015.830,-37.450,394.415,165.594,57.080,160.206
C07959=1015.836,-37.174,394.402,165.597,57.072,160.205
C07960=1015.841,-36.925,394.391,165.600,57.065,160.205
C07961=1015.846,-36.675,394.380,165.603,57.058,160.204
C07962=1015.851,-36.425,394.368,165.605,57.050,160.203
C07963=1015.856,-36.176,394.357,165.608,57.043,160.203
C07964=1015.861,-35.926,394.346,165.610,57.036,160.202
C07965=1015.866,-35.676,394.334,165.613,57.029,160.201
C07966=1015.871,-35.426,394.323,165.616,57.021,160.200
C07967=1015.877,-35.177,394.312,165.619,57.014,160.200
C07968=1015.882,-34.927,394.300,165.621,57.006,160.199
C07969=1015.887,-34.677,394.289,165.624,57.000,160.198
C07970=1015.892,-34.427,394.277,165.627,56.992,160.198
C07971=1015.897,-34.177,394.266,165.630,56.985,160.197
C07972=1015.903,-33.928,394.255,165.632,56.977,160.196
C07973=1015.908,-33.678,394.244,165.635,56.970,160.196
C07974=1015.913,-33.428,394.232,165.637,56.963,160.195
C07975=1015.918,-33.179,394.220,165.640,56.956,160.194
C07976=1015.924,-32.930,394.209,165.643,56.948,160.194
C07977=1015.929,-32.680,394.198,165.646,56.941,160.193
C07978=1015.934,-32.430,394.186,165.648,56.933,160.192
C07979=1015.939,-32.180,394.175,165.651,56.926,160.191
C07980=1015.944,-31.931,394.163,165.654,56.919,160.191
C07981=1015.950,-31.681,394.152,165.656,56.911,160.190
C07982=1015.955,-31.431,394.141,165.660,56.904,160.190
C07983=1015.960,-31.182,394.129,165.662,56.896,160.189
C07984=1015.965,-30.932,394.117,165.665,56.888,160.188
C07985=1015.971,-30.683,394.106,165.668,56.881,160.187
C07986=1015.976,-30.433,394.095,165.670,56.874,160.187
C07987=1015.981,-30.183,394.083,165.673,56.866,160.186
C07988=1015.986,-29.933,394.072,165.676,56.859,160.185
C07989=1015.991,-29.684,394.060,165.678,56.852,160.184
C07990=1015.997,-29.434,394.049,165.681,56.844,160.183
C07991=1016.002,-29.184,394.037,165.684,56.837,160.183
C07992=1016.007,-28.934,394.026,165.686,56.829,160.182
C07993=1016.012,-28.685,394.014,165.688,56.822,160.181
C07994=1016.018,-28.435,394.003,165.693,56.814,160.181
C07995=1016.023,-28.186,393.991,165.695,56.807,160.180
C07996=1016.028,-27.936,393.980,165.697,56.799,160.179
C07997=1016.033,-27.686,393.968,165.700,56.792,160.179
C07998=1016.039,-27.436,393.956,165.703,56.784,160.178
C07999=1016.044,-27.187,393.944,165.705,56.777,160.177
C08000=1016.049,-26.937,393.933,165.708,56.770,160.176
C08001=1016.055,-26.688,393.920,165.711,56.762,160.176
C08002=1016.060,-26.438,393.909,165.714,56.755,160.175
C08003=1016.065,-26.188,393.897,165.716,56.748,160.174
C08004=1016.070,-25.939,393.885,165.719,56.741,160.174
C08005=1016.075,-25.688,393.873,165.722,56.733,160.173
C08006=1016.080,-25.439,393.861,165.725,56.726,160.172
C08007=1016.085,-25.189,393.849,165.727,56.719,160.171
C08008=1016.090,-24.940,393.837,165.730,56.711,160.171
C08009=1016.095,-24.690,393.826,165.733,56.704,160.170
C08010=1016.101,-24.441,393.813,165.735,56.696,160.169
C08011=1016.106,-24.190,393.801,165.738,56.689,160.168
C08012=1016.111,-23.941,393.790,165.741,56.682,160.168
C08013=1016.117,-23.691,393.778,165.743,56.674,160.167
C08014=1016.122,-23.442,393.766,165.746,56.667,160.167
C08015=1016.127,-23.192,393.754,165.749,56.660,160.166
C08016=1016.133,-22.942,393.742,165.751,56.652,160.165
C08017=1016.138,-22.693,393.730,165.753,56.644,160.164
C08018=1016.143,-22.443,393.719,165.757,56.637,160.163
C08019=1016.148,-22.194,393.706,165.759,56.630,160.163
C08020=1016.153,-21.916,393.693,165.763,56.622,160.162
C08021=1016.159,-21.640,393.679,165.764,56.613,160.161
C08022=1016.165,-21.363,393.666,165.768,56.605,160.160
C08023=1016.171,-21.086,393.653,165.771,56.597,160.159
C08024=1016.176,-20.836,393.641,165.774,56.590,160.159
C08025=1016.182,-20.586,393.629,165.776,56.582,160.158
C08026=1016.187,-20.337,393.617,165.779,56.574,160.157
C08027=1016.192,-20.087,393.605,165.781,56.567,160.156
C08028=1016.197,-19.838,393.593,165.784,56.559,160.155
C08029=1016.203,-19.587,393.581,165.787,56.552,160.155
C08030=1016.208,-19.338,393.569,165.789,56.545,160.154
C08031=1016.214,-19.089,393.557,165.792,56.537,160.153
C08032=1016.219,-18.838,393.545,165.794,56.529,160.152
C08033=1016.224,-18.589,393.533,165.798,56.521,160.152
C08034=1016.229,-18.339,393.521,165.801,56.514,160.151
C08035=1016.234,-18.090,393.508,165.803,56.507,160.150
C08036=1016.240,-17.840,393.496,165.806,56.499,160.150
C08037=1016.245,-17.590,393.484,165.808,56.492,160.149
C08038=1016.250,-17.341,393.472,165.811,56.484,160.148
C08039=1016.256,-17.091,393.460,165.813,56.476,160.147
C08040=1016.261,-16.841,393.448,165.816,56.469,160.146
C08041=1016.266,-16.592,393.436,165.819,56.462,160.146
C08042=1016.272,-16.342,393.424,165.822,56.454,160.145
C08043=1016.277,-16.092,393.412,165.825,56.446,160.144
C08044=1016.282,-15.843,393.399,165.828,56.439,160.143
C08045=1016.288,-15.593,393.387,165.830,56.431,160.143
C08046=1016.293,-15.344,393.375,165.833,56.424,160.142
C08047=1016.298,-15.094,393.362,165.836,56.417,160.141
C08048=1016.303,-14.844,393.350,165.838,56.409,160.140
C08049=1016.308,-14.594,393.337,165.841,56.401,160.140
C08050=1016.313,-14.345,393.325,165.844,56.394,160.139
C08051=1016.319,-14.095,393.312,165.846,56.387,160.138
C08052=1016.324,-13.846,393.300,165.849,56.379,160.137
C08053=1016.330,-13.596,393.287,165.851,56.372,160.137
C08054=1016.335,-13.347,393.275,165.854,56.365,160.136
C08055=1016.339,-13.097,393.262,165.857,56.357,160.135
C08056=1016.345,-12.847,393.250,165.859,56.350,160.134
C08057=1016.350,-12.598,393.238,165.862,56.342,160.134
C08058=1016.355,-12.348,393.225,165.864,56.334,160.133
C08059=1016.361,-12.098,393.213,165.867,56.328,160.132
C08060=1016.365,-11.849,393.200,165.870,56.320,160.131
C08061=1016.371,-11.599,393.187,165.872,56.312,160.130
C08062=1016.377,-11.350,393.175,165.875,56.305,160.130
C08063=1016.382,-11.100,393.162,165.878,56.297,160.129
C08064=1016.387,-10.850,393.150,165.880,56.290,160.128
C08065=1016.392,-10.601,393.138,165.883,56.283,160.127
C08066=1016.398,-10.351,393.125,165.886,56.275,160.127
C08067=1016.403,-10.102,393.112,165.888,56.268,160.126
C08068=1016.409,-9.852,393.100,165.891,56.260,160.125
C08069=1016.413,-9.602,393.087,165.893,56.252,160.124
C08070=1016.419,-9.353,393.074,165.896,56.245,160.123
C08071=1016.424,-9.103,393.062,165.898,56.237,160.123
C08072=1016.430,-8.853,393.049,165.901,56.230,160.122
C08073=1016.435,-8.604,393.037,165.904,56.222,160.121
C08074=1016.440,-8.354,393.024,165.907,56.214,160.120
C08075=1016.446,-8.105,393.012,165.910,56.206,160.119
C08076=1016.451,-7.855,392.999,165.913,56.200,160.119
C08077=1016.456,-7.605,392.986,165.915,56.192,160.118
C08078=1016.461,-7.356,392.974,165.918,56.184,160.117
C08079=1016.467,-7.106,392.961,165.920,56.177,160.116
C08080=1016.472,-6.857,392.949,165.923,56.169,160.116
C08081=1016.478,-6.607,392.936,165.925,56.162,160.115
C08082=1016.482,-6.357,392.923,165.928,56.154,160.114
C08083=1016.488,-6.107,392.911,165.930,56.147,160.113
C08084=1016.494,-5.829,392.897,165.934,56.138,160.112
C08085=1016.500,-5.550,392.883,165.937,56.129,160.111
C08086=1016.506,-5.271,392.868,165.940,56.120,160.110
C08087=1016.512,-4.992,392.854,165.943,56.112,160.109
C08088=1016.517,-4.743,392.841,165.945,56.104,160.109
C08089=1016.523,-4.493,392.829,165.948,56.097,160.108
C08090=1016.528,-4.242,392.816,165.950,56.089,160.107
C08091=1016.534,-3.994,392.803,165.953,56.081,160.106
C08092=1016.539,-3.744,392.790,165.956,56.075,160.106
C08093=1016.543,-3.494,392.777,165.959,56.067,160.105
C08094=1016.549,-3.245,392.763,165.961,56.060,160.104
C08095=1016.554,-2.995,392.751,165.964,56.052,160.103
C08096=1016.559,-2.745,392.738,165.966,56.044,160.102
C08097=1016.564,-2.496,392.724,165.969,56.038,160.102
C08098=1016.569,-2.246,392.711,165.972,56.030,160.101
C08099=1016.575,-1.996,392.699,165.975,56.022,160.100
C08100=1016.580,-1.747,392.685,165.977,56.015,160.099
C08101=1016.585,-1.497,392.672,165.980,56.007,160.098
C08102=1016.590,-1.248,392.659,165.982,56.000,160.098
C08103=1016.596,-0.998,392.646,165.985,55.992,160.097
C08104=1016.601,-0.748,392.633,165.987,55.985,160.096
C08105=1016.606,-0.499,392.619,165.989,55.978,160.095
C08106=1016.611,-0.249,392.606,165.992,55.971,160.094
C08107=1016.617,-0.000,392.594,165.995,55.963,160.094
C08108=1016.622,0.250,392.580,165.997,55.956,160.093
C08109=1016.627,0.500,392.567,166.000,55.948,160.092
C08110=1016.632,0.749,392.553,166.002,55.941,160.091
C08111=1016.638,0.998,392.541,166.005,55.933,160.090
C08112=1016.643,1.249,392.528,166.008,55.925,160.090
C08113=1016.648,1.498,392.514,166.010,55.918,160.089
C08114=1016.653,1.748,392.501,166.013,55.910,160.088
C08115=1016.659,1.996,392.488,166.016,55.902,160.087
C08116=1016.664,2.247,392.475,166.019,55.895,160.086
C08117=1016.669,2.496,392.461,166.022,55.887,160.086
C08118=1016.674,2.746,392.448,166.024,55.880,160.085
C08119=1016.679,2.995,392.434,166.027,55.872,160.084
C08120=1016.685,3.245,392.422,166.029,55.865,160.083
C08121=1016.690,3.494,392.408,166.032,55.857,160.082
C08122=1016.695,3.744,392.395,166.035,55.850,160.082
C08123=1016.701,3.994,392.382,166.037,55.842,160.081
C08124=1016.706,4.243,392.369,166.040,55.835,160.080
C08125=1016.711,4.493,392.356,166.042,55.827,160.079
C08126=1016.717,4.743,392.342,166.045,55.820,160.078
C08127=1016.722,4.992,392.328,166.048,55.812,160.077
C08128=1016.728,5.241,392.316,166.050,55.804,160.077
C08129=1016.733,5.491,392.302,166.053,55.797,160.076
C08130=1016.738,5.741,392.289,166.055,55.789,160.075
C08131=1016.743,5.990,392.276,166.058,55.782,160.074
C08132=1016.749,6.240,392.263,166.060,55.774,160.073
C08133=1016.755,6.489,392.249,166.063,55.766,160.072
C08134=1016.760,6.740,392.236,166.065,55.759,160.071
C08135=1016.765,6.989,392.223,166.068,55.751,160.071
C08136=1016.770,7.239,392.209,166.071,55.744,160.070
C08137=1016.776,7.488,392.196,166.074,55.736,160.069
C08138=1016.781,7.738,392.182,166.077,55.728,160.068
C08139=1016.786,7.987,392.169,166.079,55.721,160.068
C08140=1016.791,8.237,392.156,166.082,55.712,160.066
C08141=1016.797,8.487,392.143,166.084,55.705,160.066
C08142=1016.803,8.736,392.129,166.087,55.697,160.065
C08143=1016.808,8.985,392.116,166.089,55.690,160.064
C08144=1016.813,9.235,392.103,166.092,55.682,160.063
C08145=1016.818,9.485,392.089,166.094,55.674,160.062
C08146=1016.825,9.734,392.075,166.097,55.667,160.061
C08147=1016.830,9.984,392.062,166.099,55.659,160.060
C08148=1016.836,10.265,392.047,166.103,55.650,160.060
C08149=1016.842,10.546,392.032,166.106,55.642,160.059
C08150=1016.848,10.826,392.017,166.109,55.633,160.058
C08151=1016.854,11.107,392.002,166.112,55.624,160.057
C08152=1016.860,11.357,391.988,166.114,55.616,160.056
C08153=1016.865,11.605,391.975,166.117,55.609,160.055
C08154=1016.870,11.856,391.962,166.119,55.601,160.054
C08155=1016.875,12.105,391.948,166.122,55.593,160.053
C08156=1016.881,12.355,391.934,166.124,55.586,160.052
C08157=1016.887,12.605,391.921,166.128,55.578,160.052
C08158=1016.892,12.854,391.908,166.131,55.570,160.051
C08159=1016.897,13.103,391.894,166.133,55.562,160.050
C08160=1016.903,13.353,391.880,166.135,55.554,160.049
C08161=1016.908,13.603,391.867,166.138,55.547,160.048
C08162=1016.913,13.853,391.853,166.141,55.539,160.047
C08163=1016.919,14.102,391.839,166.143,55.532,160.046
C08164=1016.924,14.352,391.825,166.146,55.524,160.046
C08165=1016.930,14.601,391.812,166.148,55.516,160.045
C08166=1016.935,14.851,391.798,166.151,55.509,160.044
C08167=1016.940,15.100,391.784,166.153,55.501,160.043
C08168=1016.945,15.350,391.770,166.156,55.494,160.042
C08169=1016.950,15.600,391.757,166.159,55.486,160.041
C08170=1016.955,15.849,391.743,166.161,55.479,160.040
C08171=1016.961,16.099,391.729,166.164,55.471,160.040
C08172=1016.966,16.349,391.715,166.166,55.463,160.039
C08173=1016.972,16.598,391.701,166.169,55.456,160.038
C08174=1016.977,16.848,391.687,166.171,55.448,160.037
C08175=1016.983,17.097,391.673,166.174,55.441,160.036
C08176=1016.988,17.346,391.660,166.177,55.433,160.035
C08177=1016.993,17.596,391.646,166.179,55.425,160.034
C08178=1016.999,17.845,391.632,166.182,55.418,160.033
C08179=1017.004,18.095,391.618,166.184,55.410,160.033
C08180=1017.010,18.344,391.604,166.187,55.403,160.032
C08181=1017.015,18.594,391.591,166.189,55.394,160.031
C08182=1017.020,18.844,391.576,166.192,55.387,160.030
C08183=1017.025,19.093,391.562,166.194,55.379,160.029
C08184=1017.031,19.343,391.548,166.197,55.372,160.028
C08185=1017.036,19.593,391.535,166.200,55.364,160.027
C08186=1017.042,19.842,391.521,166.202,55.356,160.026
C08187=1017.047,20.092,391.506,166.205,55.349,160.026
C08188=1017.052,20.342,391.492,166.207,55.341,160.025
C08189=1017.058,20.591,391.478,166.210,55.334,160.024
C08190=1017.063,20.840,391.464,166.213,55.326,160.023
C08191=1017.068,21.090,391.449,166.215,55.319,160.022
C08192=1017.073,21.340,391.436,166.218,55.311,160.021
C08193=1017.079,21.589,391.422,166.220,55.303,160.020
C08194=1017.084,21.838,391.408,166.223,55.296,160.020
C08195=1017.089,22.088,391.394,166.226,55.288,160.019
C08196=1017.094,22.338,391.380,166.229,55.280,160.018
C08197=1017.100,22.586,391.365,166.232,55.272,160.017
C08198=1017.105,22.836,391.351,166.234,55.265,160.016
C08199=1017.111,23.086,391.338,166.237,55.257,160.016
C08200=1017.115,23.336,391.323,166.239,55.249,160.014
C08201=1017.121,23.585,391.309,166.242,55.242,160.014
C08202=1017.126,23.835,391.295,166.245,55.234,160.013
C08203=1017.132,24.084,391.281,166.247,55.227,160.012
C08204=1017.137,24.334,391.266,166.249,55.219,160.011
C08205=1017.143,24.584,391.252,166.252,55.211,160.010
C08206=1017.149,24.833,391.238,166.255,55.204,160.009
C08207=1017.154,25.082,391.224,166.257,55.196,160.008
C08208=1017.159,25.332,391.209,166.260,55.188,160.007
C08209=1017.165,25.582,391.195,166.262,55.181,160.007
C08210=1017.170,25.831,391.182,166.265,55.173,160.006
C08211=1017.175,26.081,391.168,166.267,55.165,160.005
C08212=1017.181,26.363,391.151,166.271,55.157,160.004
C08213=1017.187,26.645,391.135,166.274,55.148,160.003
C08214=1017.193,26.927,391.119,166.276,55.139,160.002
C08215=1017.200,27.210,391.102,166.279,55.131,160.001
C08216=1017.205,27.460,391.088,166.282,55.123,160.000
C08217=1017.210,27.709,391.074,166.284,55.116,159.999
C08218=1017.215,27.958,391.059,166.286,55.108,159.998
C08219=1017.221,28.208,391.045,166.289,55.100,159.997
C08220=1017.226,28.457,391.030,166.292,55.093,159.996
C08221=1017.231,28.707,391.016,166.295,55.085,159.996
C08222=1017.236,28.957,391.002,166.297,55.077,159.995
C08223=1017.242,29.206,390.987,166.300,55.070,159.994
C08224=1017.247,29.456,390.973,166.302,55.062,159.993
C08225=1017.252,29.704,390.958,166.305,55.055,159.992
C08226=1017.258,29.955,390.943,166.307,55.047,159.991
C08227=1017.263,30.204,390.929,166.310,55.039,159.990
C08228=1017.268,30.454,390.914,166.313,55.032,159.989
C08229=1017.274,30.703,390.900,166.315,55.024,159.989
C08230=1017.279,30.952,390.886,166.318,55.016,159.988
C08231=1017.285,31.202,390.870,166.320,55.009,159.987
C08232=1017.290,31.451,390.857,166.323,55.001,159.986
C08233=1017.295,31.701,390.842,166.325,54.993,159.985
C08234=1017.301,31.951,390.827,166.328,54.986,159.984
C08235=1017.306,32.201,390.813,166.331,54.978,159.983
C08236=1017.312,32.450,390.798,166.333,54.970,159.982
C08237=1017.317,32.699,390.783,166.336,54.963,159.981
C08238=1017.322,32.948,390.769,166.339,54.955,159.981
C08239=1017.327,33.198,390.754,166.341,54.947,159.980
C08240=1017.333,33.447,390.740,166.344,54.940,159.979
C08241=1017.338,33.697,390.725,166.346,54.932,159.978
C08242=1017.344,33.947,390.711,166.349,54.924,159.977
C08243=1017.349,34.196,390.696,166.351,54.917,159.976
C08244=1017.354,34.446,390.682,166.354,54.909,159.975
C08245=1017.359,34.695,390.666,166.356,54.901,159.974
C08246=1017.365,34.945,390.653,166.359,54.894,159.973
C08247=1017.370,35.195,390.637,166.361,54.886,159.972
C08248=1017.376,35.443,390.622,166.364,54.878,159.972
C08249=1017.381,35.693,390.608,166.366,54.870,159.970
C08250=1017.387,35.942,390.593,166.369,54.863,159.970
C08251=1017.392,36.192,390.579,166.372,54.856,159.969
C08252=1017.398,36.442,390.564,166.374,54.847,159.968
C08253=1017.403,36.691,390.549,166.377,54.840,159.967
C08254=1017.408,36.941,390.534,166.380,54.833,159.966
C08255=1017.413,37.190,390.519,166.382,54.824,159.965
C08256=1017.419,37.440,390.504,166.385,54.817,159.964
C08257=1017.424,37.690,390.490,166.387,54.810,159.964
C08258=1017.429,37.939,390.475,166.390,54.802,159.962
C08259=1017.434,38.188,390.459,166.392,54.794,159.962
C08260=1017.440,38.438,390.445,166.395,54.787,159.961
C08261=1017.445,38.688,390.430,166.398,54.779,159.960
C08262=1017.450,38.937,390.415,166.400,54.771,159.959
C08263=1017.455,39.186,390.400,166.403,54.764,159.958
C08264=1017.462,39.436,390.385,166.406,54.756,159.957
C08265=1017.467,39.685,390.370,166.408,54.748,159.956
C08266=1017.471,39.935,390.355,166.411,54.741,159.956
C08267=1017.476,40.185,390.340,166.413,54.733,159.954
C08268=1017.483,40.434,390.325,166.416,54.725,159.954
C08269=1017.488,40.683,390.310,166.419,54.718,159.953
C08270=1017.493,40.933,390.295,166.421,54.710,159.952
C08271=1017.498,41.183,390.280,166.424,54.703,159.951
C08272=1017.504,41.432,390.265,166.427,54.695,159.950
C08273=1017.509,41.682,390.250,166.429,54.687,159.949
C08274=1017.514,41.931,390.235,166.432,54.680,159.948
C08275=1017.520,42.181,390.219,166.434,54.672,159.947
C08276=1017.525,42.462,390.202,166.436,54.664,159.946
C08277=1017.531,42.745,390.185,166.440,54.655,159.945
C08278=1017.537,43.027,390.168,166.443,54.647,159.944
C08279=1017.543,43.310,390.151,166.445,54.639,159.943
C08280=1017.548,43.559,390.135,166.448,54.630,159.942
C08281=1017.553,43.808,390.120,166.450,54.623,159.942
C08282=1017.559,44.058,390.105,166.453,54.616,159.941
C08283=1017.564,44.308,390.090,166.456,54.608,159.940
C08284=1017.569,44.557,390.074,166.458,54.600,159.939
C08285=1017.575,44.807,390.059,166.460,54.593,159.938
C08286=1017.580,45.056,390.044,166.463,54.586,159.937
C08287=1017.585,45.305,390.028,166.466,54.579,159.936
C08288=1017.590,45.555,390.013,166.468,54.570,159.935
C08289=1017.595,45.805,389.998,166.471,54.563,159.934
C08290=1017.601,46.053,389.982,166.474,54.556,159.934
C08291=1017.606,46.303,389.966,166.476,54.548,159.933
C08292=1017.612,46.552,389.951,166.479,54.540,159.932
C08293=1017.617,46.802,389.936,166.482,54.533,159.931
C08294=1017.621,47.052,389.920,166.484,54.526,159.930
C08295=1017.627,47.301,389.905,166.487,54.517,159.929
C08296=1017.632,47.551,389.889,166.488,54.510,159.928
C08297=1017.637,47.801,389.874,166.491,54.503,159.927
C08298=1017.642,48.050,389.859,166.494,54.495,159.926
C08299=1017.647,48.299,389.844,166.496,54.488,159.926
C08300=1017.653,48.548,389.827,166.499,54.480,159.925
C08301=1017.658,48.798,389.812,166.502,54.472,159.924
C08302=1017.664,49.048,389.797,166.504,54.465,159.923
C08303=1017.669,49.297,389.781,166.507,54.457,159.922
C08304=1017.674,49.546,389.766,166.510,54.450,159.921
C08305=1017.680,49.796,389.751,166.512,54.442,159.920
C08306=1017.685,50.045,389.736,166.515,54.434,159.919
C08307=1017.691,50.295,389.719,166.518,54.427,159.918
C08308=1017.696,50.544,389.704,166.520,54.419,159.917
C08309=1017.701,50.793,389.689,166.523,54.411,159.917
C08310=1017.706,51.043,389.673,166.526,54.404,159.916
C08311=1017.711,51.293,389.658,166.527,54.396,159.915
C08312=1017.717,51.542,389.642,166.530,54.389,159.914
C08313=1017.722,51.791,389.626,166.532,54.381,159.913
C08314=1017.727,52.041,389.611,166.535,54.374,159.912
C08315=1017.732,52.291,389.595,166.537,54.366,159.911
C08316=1017.737,52.540,389.580,166.540,54.358,159.910
C08317=1017.743,52.789,389.564,166.543,54.350,159.909
C08318=1017.748,53.039,389.549,166.545,54.343,159.908
C08319=1017.754,53.289,389.533,166.548,54.336,159.907
C08320=1017.759,53.538,389.518,166.551,54.327,159.906
C08321=1017.765,53.787,389.502,166.553,54.320,159.906
C08322=1017.770,54.036,389.487,166.556,54.312,159.905
C08323=1017.776,54.286,389.471,166.559,54.305,159.904
C08324=1017.781,54.536,389.456,166.561,54.297,159.903
C08325=1017.787,54.785,389.440,166.564,54.289,159.902
C08326=1017.792,55.034,389.425,166.566,54.281,159.901
C08327=1017.797,55.284,389.409,166.569,54.274,159.900
C08328=1017.803,55.533,389.393,166.571,54.266,159.899
C08329=1017.808,55.783,389.377,166.574,54.258,159.898
C08330=1017.813,56.032,389.362,166.577,54.251,159.897
C08331=1017.819,56.282,389.346,166.579,54.243,159.896
C08332=1017.824,56.531,389.330,166.582,54.235,159.895
C08333=1017.829,56.781,389.315,166.584,54.227,159.894
C08334=1017.834,57.030,389.300,166.587,54.220,159.893
C08335=1017.840,57.280,389.283,166.590,54.212,159.892
C08336=1017.845,57.529,389.268,166.592,54.205,159.892
C08337=1017.851,57.779,389.253,166.595,54.197,159.891
C08338=1017.856,58.028,389.237,166.597,54.188,159.890
C08339=1017.862,58.277,389.221,166.600,54.181,159.889
C08340=1017.868,58.559,389.203,166.603,54.172,159.888
C08341=1017.874,58.842,389.186,166.606,54.164,159.887
C08342=1017.880,59.124,389.167,166.609,54.155,159.886
C08343=1017.886,59.406,389.150,166.612,54.145,159.884
C08344=1017.892,59.656,389.134,166.615,54.138,159.884
C08345=1017.897,59.905,389.119,166.618,54.130,159.883
C08346=1017.903,60.155,389.103,166.621,54.123,159.882
C08347=1017.908,60.404,389.087,166.623,54.115,159.881
C08348=1017.914,60.654,389.072,166.625,54.107,159.880
C08349=1017.919,60.902,389.056,166.628,54.099,159.879
C08350=1017.925,61.152,389.040,166.631,54.091,159.878
C08351=1017.930,61.402,389.025,166.633,54.083,159.877
C08352=1017.936,61.651,389.009,166.636,54.076,159.876
C08353=1017.941,61.901,388.993,166.638,54.068,159.875
C08354=1017.947,62.149,388.977,166.641,54.060,159.874
C08355=1017.952,62.400,388.961,166.644,54.053,159.873
C08356=1017.958,62.649,388.945,166.646,54.045,159.872
C08357=1017.963,62.898,388.930,166.648,54.037,159.871
C08358=1017.969,63.148,388.914,166.651,54.029,159.870
C08359=1017.973,63.398,388.897,166.654,54.021,159.869
C08360=1017.979,63.647,388.882,166.657,54.014,159.868
C08361=1017.985,63.896,388.865,166.659,54.006,159.867
C08362=1017.989,64.146,388.850,166.662,53.999,159.867
C08363=1017.995,64.395,388.833,166.664,53.991,159.866
C08364=1018.000,64.645,388.817,166.667,53.984,159.865
C08365=1018.005,64.894,388.801,166.670,53.976,159.864
C08366=1018.011,65.143,388.785,166.673,53.968,159.863
C08367=1018.016,65.393,388.769,166.675,53.960,159.862
C08368=1018.022,65.642,388.753,166.678,53.953,159.861
C08369=1018.027,65.892,388.736,166.680,53.945,159.860
C08370=1018.032,66.142,388.721,166.683,53.938,159.859
C08371=1018.037,66.391,388.704,166.686,53.930,159.858
C08372=1018.043,66.640,388.688,166.689,53.923,159.858
C08373=1018.049,66.889,388.672,166.691,53.915,159.856
C08374=1018.053,67.139,388.656,166.694,53.907,159.856
C08375=1018.059,67.388,388.640,166.695,53.900,159.854
C08376=1018.064,67.637,388.623,166.698,53.892,159.853
C08377=1018.070,67.887,388.607,166.701,53.884,159.853
C08378=1018.075,68.137,388.591,166.703,53.876,159.852
C08379=1018.081,68.386,388.574,166.706,53.869,159.851
C08380=1018.085,68.635,388.558,166.709,53.861,159.850
C08381=1018.091,68.885,388.542,166.712,53.854,159.849
C08382=1018.096,69.134,388.525,166.714,53.846,159.848
C08383=1018.101,69.384,388.509,166.717,53.839,159.847
C08384=1018.107,69.633,388.493,166.719,53.831,159.846
C08385=1018.112,69.883,388.476,166.722,53.823,159.845
C08386=1018.117,70.131,388.460,166.725,53.815,159.844
C08387=1018.122,70.381,388.443,166.728,53.808,159.844
C08388=1018.128,70.630,388.427,166.730,53.800,159.842
C08389=1018.133,70.879,388.410,166.733,53.793,159.842
C08390=1018.138,71.130,388.394,166.736,53.785,159.841
C08391=1018.144,71.379,388.378,166.737,53.778,159.840
C08392=1018.149,71.629,388.361,166.740,53.770,159.839
C08393=1018.154,71.878,388.345,166.743,53.763,159.838
C08394=1018.160,72.127,388.328,166.745,53.755,159.837
C08395=1018.165,72.377,388.312,166.748,53.748,159.836
C08396=1018.171,72.626,388.295,166.751,53.740,159.835
C08397=1018.175,72.875,388.279,166.754,53.732,159.834
C08398=1018.181,73.125,388.262,166.756,53.724,159.833
C08399=1018.187,73.374,388.246,166.759,53.717,159.832
C08400=1018.191,73.623,388.229,166.762,53.709,159.831
C08401=1018.196,73.873,388.212,166.764,53.701,159.830
C08402=1018.202,74.122,388.196,166.767,53.694,159.830
C08403=1018.207,74.372,388.179,166.770,53.686,159.829
C08404=1018.213,74.654,388.161,166.773,53.678,159.828
C08405=1018.219,74.936,388.143,166.775,53.669,159.826
C08406=1018.226,75.218,388.124,166.779,53.661,159.826
C08407=1018.232,75.500,388.104,166.782,53.652,159.824
C08408=1018.237,75.750,388.088,166.784,53.644,159.823
C08409=1018.243,75.999,388.071,166.787,53.637,159.823
C08410=1018.247,76.248,388.055,166.790,53.629,159.822
C08411=1018.253,76.498,388.038,166.793,53.621,159.821
C08412=1018.258,76.747,388.021,166.795,53.613,159.820
C08413=1018.264,76.997,388.005,166.798,53.606,159.819
C08414=1018.269,77.246,387.988,166.801,53.598,159.818
C08415=1018.274,77.495,387.972,166.802,53.591,159.817
C08416=1018.279,77.745,387.955,166.805,53.583,159.816
C08417=1018.284,77.994,387.938,166.808,53.576,159.815
C08418=1018.290,78.244,387.920,166.810,53.568,159.814
C08419=1018.295,78.493,387.903,166.813,53.561,159.813
C08420=1018.299,78.742,387.887,166.816,53.553,159.812
C08421=1018.305,78.991,387.871,166.819,53.546,159.811
C08422=1018.311,79.241,387.853,166.821,53.538,159.810
C08423=1018.316,79.490,387.836,166.824,53.531,159.810
C08424=1018.321,79.740,387.819,166.827,53.523,159.809
C08425=1018.326,79.989,387.803,166.829,53.516,159.808
C08426=1018.331,80.238,387.786,166.831,53.508,159.807
C08427=1018.337,80.487,387.768,166.834,53.501,159.806
C08428=1018.342,80.737,387.752,166.837,53.493,159.805
C08429=1018.347,80.987,387.735,166.840,53.486,159.804
C08430=1018.352,81.236,387.718,166.842,53.478,159.803
C08431=1018.358,81.486,387.700,166.845,53.471,159.802
C08432=1018.363,81.735,387.684,166.848,53.463,159.801
C08433=1018.368,81.984,387.667,166.851,53.455,159.800
C08434=1018.374,82.233,387.650,166.853,53.447,159.799
C08435=1018.379,82.483,387.633,166.856,53.440,159.799
C08436=1018.384,82.732,387.616,166.859,53.432,159.798
C08437=1018.389,82.982,387.599,166.861,53.424,159.797
C08438=1018.395,83.231,387.582,166.864,53.417,159.796
C08439=1018.400,83.481,387.565,166.866,53.410,159.795
C08440=1018.405,83.730,387.548,166.869,53.402,159.794
C08441=1018.410,83.979,387.531,166.872,53.395,159.793
C08442=1018.416,84.228,387.514,166.875,53.387,159.792
C08443=1018.421,84.478,387.497,166.877,53.379,159.791
C08444=1018.426,84.727,387.480,166.880,53.372,159.790
C08445=1018.431,84.977,387.463,166.883,53.364,159.789
C08446=1018.437,85.226,387.446,166.885,53.356,159.788
C08447=1018.442,85.475,387.428,166.888,53.349,159.787
C08448=1018.447,85.725,387.412,166.891,53.341,159.786
C08449=1018.454,85.974,387.395,166.893,53.333,159.785
C08450=1018.459,86.223,387.378,166.896,53.326,159.785
C08451=1018.464,86.473,387.361,166.899,53.318,159.784
C08452=1018.470,86.722,387.343,166.901,53.310,159.782
C08453=1018.475,86.972,387.327,166.904,53.303,159.782
C08454=1018.480,87.221,387.309,166.907,53.295,159.781
C08455=1018.485,87.470,387.292,166.910,53.288,159.780
C08456=1018.490,87.719,387.276,166.913,53.280,159.779
C08457=1018.496,87.968,387.258,166.915,53.272,159.778
C08458=1018.501,88.218,387.241,166.918,53.265,159.777
C08459=1018.506,88.467,387.224,166.921,53.257,159.776
C08460=1018.512,88.717,387.207,166.923,53.249,159.775
C08461=1018.517,88.966,387.189,166.926,53.242,159.774
C08462=1018.522,89.215,387.172,166.929,53.234,159.773
C08463=1018.528,89.464,387.155,166.932,53.227,159.772
C08464=1018.532,89.714,387.137,166.934,53.219,159.771
C08465=1018.538,89.963,387.120,166.937,53.212,159.771
C08466=1018.543,90.213,387.103,166.940,53.204,159.770
C08467=1018.549,90.462,387.085,166.942,53.197,159.769
C08468=1018.554,90.745,387.065,166.945,53.188,159.768
C08469=1018.561,91.027,387.045,166.949,53.180,159.767
C08470=1018.566,91.309,387.026,166.952,53.171,159.766
C08471=1018.573,91.591,387.006,166.955,53.163,159.765
C08472=1018.578,91.871,386.986,166.958,53.154,159.763
C08473=1018.584,92.150,386.967,166.961,53.146,159.763
C08474=1018.589,92.400,386.949,166.963,53.139,159.761
C08475=1018.594,92.649,386.932,166.966,53.131,159.761
C08476=1018.600,92.898,386.915,166.968,53.124,159.760
C08477=1018.605,93.147,386.897,166.971,53.116,159.759
C08478=1018.610,93.397,386.879,166.974,53.109,159.758
C08479=1018.615,93.646,386.862,166.977,53.101,159.757
C08480=1018.621,93.895,386.845,166.980,53.094,159.756
C08481=1018.626,94.144,386.827,166.982,53.086,159.755
C08482=1018.631,94.394,386.809,166.985,53.078,159.754
C08483=1018.636,94.643,386.792,166.988,53.071,159.753
C08484=1018.642,94.893,386.774,166.991,53.063,159.752
C08485=1018.648,95.142,386.757,166.994,53.056,159.751
C08486=1018.652,95.392,386.739,166.996,53.048,159.750
C08487=1018.658,95.641,386.722,166.999,53.041,159.750
C08488=1018.663,95.890,386.704,167.002,53.033,159.749
C08489=1018.668,96.140,386.686,167.005,53.025,159.747
C08490=1018.674,96.389,386.668,167.008,53.018,159.747
C08491=1018.679,96.638,386.651,167.010,53.010,159.746
C08492=1018.684,96.887,386.634,167.013,53.003,159.745
C08493=1018.689,97.137,386.616,167.016,52.995,159.744
C08494=1018.695,97.386,386.598,167.018,52.987,159.743
C08495=1018.700,97.635,386.581,167.022,52.980,159.742
C08496=1018.705,97.884,386.564,167.024,52.972,159.741
C08497=1018.711,98.135,386.545,167.027,52.964,159.740
C08498=1018.716,98.384,386.528,167.030,52.957,159.739
C08499=1018.722,98.633,386.510,167.032,52.949,159.738
C08500=1018.727,98.882,386.493,167.035,52.941,159.737
C08501=1018.732,99.132,386.475,167.038,52.934,159.736
C08502=1018.737,99.381,386.458,167.041,52.926,159.735
C08503=1018.742,99.630,386.439,167.044,52.919,159.735
C08504=1018.748,99.880,386.421,167.045,52.912,159.733
C08505=1018.753,100.129,386.403,167.049,52.905,159.733
C08506=1018.758,100.378,386.385,167.051,52.897,159.732
C08507=1018.763,100.628,386.368,167.054,52.890,159.731
C08508=1018.768,100.877,386.349,167.057,52.882,159.730
C08509=1018.774,101.126,386.332,167.060,52.875,159.729
C08510=1018.778,101.375,386.314,167.063,52.867,159.728
C08511=1018.784,101.625,386.296,167.066,52.860,159.727
C08512=1018.789,101.874,386.278,167.068,52.852,159.726
C08513=1018.795,102.123,386.260,167.071,52.845,159.725
C08514=1018.799,102.373,386.242,167.074,52.837,159.724
C08515=1018.804,102.622,386.224,167.077,52.830,159.724
C08516=1018.810,102.871,386.206,167.080,52.822,159.723
C08517=1018.815,103.120,386.188,167.082,52.814,159.722
C08518=1018.821,103.370,386.170,167.086,52.807,159.721
C08519=1018.825,103.620,386.152,167.087,52.800,159.720
C08520=1018.831,103.869,386.134,167.090,52.792,159.719
C08521=1018.836,104.117,386.115,167.093,52.785,159.718
C08522=1018.842,104.366,386.098,167.096,52.778,159.717
C08523=1018.847,104.616,386.079,167.099,52.770,159.716
C08524=1018.852,104.866,386.061,167.101,52.762,159.715
C08525=1018.857,105.115,386.044,167.104,52.755,159.714
C08526=1018.862,105.364,386.025,167.107,52.747,159.713
C08527=1018.868,105.613,386.008,167.110,52.740,159.713
C08528=1018.873,105.863,385.989,167.113,52.732,159.712
C08529=1018.878,106.112,385.972,167.116,52.725,159.711
C08530=1018.886,106.504,385.943,167.121,52.713,159.709
C08531=1018.895,106.896,385.915,167.125,52.701,159.708
C08532=1018.903,107.288,385.886,167.130,52.689,159.706
C08533=1018.911,107.680,385.858,167.134,52.677,159.705
C08534=1018.917,107.928,385.839,167.137,52.670,159.704
C08535=1018.922,108.178,385.821,167.139,52.662,159.703
C08536=1018.928,108.427,385.803,167.142,52.655,159.702
C08537=1018.932,108.677,385.785,167.145,52.647,159.701
C08538=1018.938,108.926,385.767,167.148,52.639,159.700
C08539=1018.944,109.175,385.748,167.151,52.632,159.699
C08540=1018.948,109.425,385.730,167.154,52.624,159.698
C08541=1018.954,109.674,385.712,167.157,52.617,159.698
C08542=1018.959,109.924,385.694,167.159,52.609,159.697
C08543=1018.964,110.172,385.675,167.162,52.601,159.695
C08544=1018.969,110.422,385.657,167.165,52.594,159.695
C08545=1018.975,110.671,385.639,167.168,52.587,159.694
C08546=1018.980,110.920,385.620,167.171,52.579,159.693
C08547=1018.985,111.170,385.602,167.174,52.572,159.692
C08548=1018.990,111.419,385.584,167.177,52.565,159.691
C08549=1018.996,111.667,385.565,167.180,52.557,159.690
C08550=1019.001,111.917,385.547,167.182,52.549,159.689
C08551=1019.006,112.167,385.529,167.185,52.542,159.688
C08552=1019.011,112.416,385.510,167.188,52.534,159.687
C08553=1019.016,112.666,385.491,167.191,52.527,159.687
C08554=1019.021,112.914,385.473,167.194,52.520,159.686
C08555=1019.026,113.164,385.454,167.197,52.512,159.685
C08556=1019.032,113.413,385.435,167.200,52.505,159.684
C08557=1019.037,113.662,385.417,167.202,52.498,159.683
C08558=1019.042,113.911,385.398,167.205,52.491,159.682
C08559=1019.047,114.161,385.380,167.208,52.483,159.681
C08560=1019.052,114.410,385.361,167.211,52.476,159.680
C08561=1019.057,114.659,385.342,167.214,52.469,159.679
C08562=1019.063,114.909,385.323,167.217,52.461,159.678
C08563=1019.068,115.157,385.304,167.220,52.454,159.678
C08564=1019.073,115.407,385.286,167.223,52.446,159.677
C08565=1019.078,115.656,385.267,167.226,52.439,159.676
C08566=1019.082,115.906,385.248,167.228,52.431,159.675
C08567=1019.087,116.155,385.229,167.232,52.424,159.674
C08568=1019.093,116.404,385.210,167.234,52.416,159.673
C08569=1019.098,116.653,385.192,167.238,52.409,159.672
C08570=1019.103,116.902,385.173,167.240,52.402,159.671
C08571=1019.108,117.152,385.155,167.243,52.395,159.670
C08572=1019.113,117.401,385.136,167.246,52.387,159.669
C08573=1019.118,117.650,385.117,167.249,52.380,159.669
C08574=1019.124,117.900,385.098,167.252,52.372,159.668
C08575=1019.129,118.148,385.079,167.254,52.365,159.667
C08576=1019.135,118.398,385.060,167.257,52.358,159.666
C08577=1019.139,118.647,385.042,167.260,52.350,159.665
C08578=1019.144,118.896,385.023,167.263,52.343,159.664
C08579=1019.150,119.145,385.004,167.266,52.336,159.663
C08580=1019.155,119.395,384.986,167.269,52.328,159.662
C08581=1019.161,119.644,384.966,167.272,52.321,159.661
C08582=1019.166,119.893,384.948,167.275,52.313,159.660
C08583=1019.170,120.143,384.929,167.278,52.306,159.660
C08584=1019.175,120.392,384.910,167.280,52.298,159.659
C08585=1019.181,120.641,384.891,167.284,52.291,159.658
C08586=1019.186,120.891,384.872,167.286,52.284,159.657
C08587=1019.191,121.140,384.853,167.289,52.276,159.656
C08588=1019.196,121.388,384.834,167.293,52.268,159.655
C08589=1019.202,121.638,384.815,167.296,52.261,159.654
C08590=1019.207,121.887,384.797,167.299,52.254,159.653
C08591=1019.212,122.136,384.778,167.302,52.246,159.652
C08592=1019.217,122.385,384.759,167.305,52.239,159.652
C08593=1019.223,122.635,384.740,167.308,52.231,159.651
C08594=1019.228,122.917,384.718,167.311,52.222,159.649
C08595=1019.235,123.200,384.697,167.314,52.215,159.648
C08596=1019.240,123.482,384.675,167.317,52.206,159.647
C08597=1019.246,123.764,384.654,167.321,52.198,159.646
C08598=1019.252,124.014,384.636,167.324,52.190,159.645
C08599=1019.257,124.262,384.617,167.327,52.183,159.645
C08600=1019.263,124.512,384.597,167.330,52.175,159.644
C08601=1019.267,124.761,384.578,167.333,52.168,159.643
C08602=1019.273,125.010,384.559,167.336,52.160,159.642
C08603=1019.277,125.260,384.541,167.340,52.152,159.641
C08604=1019.283,125.509,384.521,167.343,52.145,159.640
C08605=1019.288,125.758,384.502,167.346,52.138,159.639
C08606=1019.294,126.007,384.483,167.348,52.130,159.638
C08607=1019.300,126.257,384.464,167.352,52.123,159.637
C08608=1019.305,126.505,384.445,167.354,52.115,159.636
C08609=1019.310,126.755,384.426,167.357,52.107,159.635
C08610=1019.315,127.004,384.408,167.360,52.100,159.635
C08611=1019.321,127.254,384.388,167.363,52.093,159.634
C08612=1019.326,127.502,384.370,167.366,52.086,159.633
C08613=1019.332,127.752,384.350,167.369,52.078,159.632
C08614=1019.336,128.001,384.331,167.373,52.070,159.631
C08615=1019.342,128.250,384.312,167.376,52.063,159.630
C08616=1019.347,128.500,384.292,167.379,52.055,159.629
C08617=1019.352,128.748,384.273,167.382,52.048,159.628
C08618=1019.358,128.998,384.254,167.385,52.041,159.627
C08619=1019.363,129.247,384.235,167.388,52.033,159.626
C08620=1019.369,129.496,384.216,167.391,52.025,159.625
C08621=1019.374,129.745,384.198,167.395,52.018,159.625
C08622=1019.379,129.995,384.178,167.398,52.010,159.624
C08623=1019.385,130.244,384.158,167.401,52.003,159.623
C08624=1019.390,130.493,384.139,167.404,51.995,159.622
C08625=1019.395,130.742,384.119,167.407,51.988,159.621
C08626=1019.400,130.992,384.100,167.410,51.981,159.620
C08627=1019.405,131.241,384.081,167.413,51.974,159.619
C08628=1019.410,131.490,384.061,167.416,51.966,159.618
C08629=1019.415,131.739,384.042,167.419,51.959,159.618
C08630=1019.420,131.989,384.023,167.422,51.951,159.617
C08631=1019.426,132.238,384.003,167.425,51.944,159.616
C08632=1019.431,132.487,383.983,167.428,51.937,159.615
C08633=1019.436,132.736,383.964,167.431,51.930,159.614
C08634=1019.441,132.985,383.945,167.434,51.922,159.613
C08635=1019.446,133.235,383.925,167.437,51.915,159.612
C08636=1019.452,133.484,383.905,167.440,51.907,159.611
C08637=1019.457,133.732,383.886,167.443,51.900,159.610
C08638=1019.462,133.982,383.866,167.447,51.892,159.610
C08639=1019.467,134.232,383.847,167.450,51.885,159.609
C08640=1019.473,134.480,383.828,167.453,51.878,159.608
C08641=1019.478,134.729,383.807,167.456,51.871,159.607
C08642=1019.483,134.979,383.788,167.459,51.863,159.606
C08643=1019.488,135.228,383.769,167.462,51.856,159.605
C08644=1019.494,135.477,383.749,167.465,51.848,159.604
C08645=1019.499,135.727,383.729,167.468,51.841,159.603
C08646=1019.504,135.975,383.710,167.471,51.834,159.602
C08647=1019.509,136.225,383.690,167.474,51.827,159.602
C08648=1019.515,136.474,383.670,167.477,51.819,159.601
C08649=1019.519,136.723,383.651,167.481,51.812,159.600
C08650=1019.525,136.972,383.632,167.484,51.804,159.599
C08651=1019.530,137.221,383.611,167.488,51.797,159.598
C08652=1019.535,137.470,383.592,167.490,51.789,159.597
C08653=1019.540,137.720,383.572,167.494,51.782,159.596
C08654=1019.546,137.969,383.552,167.496,51.775,159.595
C08655=1019.550,138.218,383.533,167.500,51.768,159.595
C08656=1019.556,138.467,383.512,167.503,51.760,159.594
C08657=1019.561,138.716,383.493,167.506,51.753,159.593
C08658=1019.567,138.999,383.470,167.509,51.744,159.592
C08659=1019.573,139.281,383.447,167.513,51.736,159.591
C08660=1019.579,139.563,383.426,167.517,51.728,159.590
C08661=1019.585,139.846,383.403,167.520,51.720,159.589
C08662=1019.589,140.094,383.383,167.524,51.713,159.588
C08663=1019.594,140.344,383.363,167.527,51.705,159.587
C08664=1019.600,140.593,383.343,167.530,51.698,159.586
C08665=1019.605,140.842,383.323,167.533,51.690,159.585
C08666=1019.610,141.091,383.303,167.537,51.683,159.585
C08667=1019.616,141.340,383.284,167.540,51.676,159.584
C08668=1019.621,141.589,383.263,167.543,51.669,159.583
C08669=1019.626,141.839,383.243,167.546,51.661,159.582
C08670=1019.631,142.088,383.223,167.549,51.654,159.581
C08671=1019.636,142.337,383.204,167.552,51.646,159.580
C08672=1019.642,142.586,383.183,167.555,51.639,159.579
C08673=1019.647,142.835,383.163,167.559,51.632,159.578
C08674=1019.652,143.084,383.144,167.563,51.624,159.578
C08675=1019.657,143.333,383.123,167.566,51.618,159.577
C08676=1019.662,143.583,383.103,167.569,51.610,159.576
C08677=1019.667,143.832,383.083,167.572,51.603,159.575
C08678=1019.673,144.081,383.063,167.575,51.595,159.574
C08679=1019.678,144.330,383.043,167.578,51.588,159.573
C08680=1019.683,144.579,383.023,167.582,51.580,159.572
C08681=1019.689,144.828,383.004,167.585,51.573,159.572
C08682=1019.694,145.078,382.983,167.588,51.566,159.571
C08683=1019.699,145.327,382.962,167.591,51.559,159.570
C08684=1019.704,145.576,382.943,167.594,51.551,159.569
C08685=1019.709,145.825,382.923,167.598,51.544,159.568
C08686=1019.715,146.074,382.903,167.602,51.536,159.567
C08687=1019.720,146.323,382.882,167.605,51.529,159.566
C08688=1019.725,146.573,382.862,167.608,51.523,159.566
C08689=1019.730,146.822,382.842,167.611,51.515,159.565
C08690=1019.735,147.071,382.821,167.614,51.508,159.564
C08691=1019.740,147.319,382.801,167.617,51.500,159.563
C08692=1019.745,147.568,382.780,167.620,51.493,159.562
C08693=1019.750,147.818,382.760,167.624,51.485,159.561
C08694=1019.756,148.067,382.740,167.628,51.479,159.560
C08695=1019.762,148.316,382.720,167.631,51.472,159.560
C08696=1019.767,148.565,382.699,167.634,51.464,159.559
C08697=1019.772,148.814,382.679,167.637,51.457,159.558
C08698=1019.777,149.063,382.658,167.640,51.449,159.557
C08699=1019.782,149.312,382.639,167.644,51.442,159.556
C08700=1019.787,149.562,382.618,167.648,51.435,159.555
C08701=1019.792,149.811,382.598,167.651,51.428,159.554
C08702=1019.797,150.060,382.577,167.654,51.421,159.554
C08703=1019.803,150.309,382.557,167.657,51.414,159.553
C08704=1019.808,150.558,382.536,167.660,51.406,159.552
C08705=1019.813,150.807,382.515,167.664,51.399,159.551
C08706=1019.818,151.056,382.495,167.667,51.391,159.550
C08707=1019.824,151.305,382.474,167.671,51.385,159.549
C08708=1019.829,151.555,382.454,167.674,51.378,159.549
C08709=1019.834,151.804,382.433,167.677,51.370,159.548
C08710=1019.839,152.053,382.413,167.681,51.363,159.547
C08711=1019.845,152.302,382.392,167.684,51.355,159.546
C08712=1019.849,152.550,382.372,167.687,51.348,159.545
C08713=1019.855,152.799,382.351,167.690,51.341,159.544
C08714=1019.860,153.049,382.331,167.694,51.334,159.543
C08715=1019.865,153.298,382.310,167.698,51.327,159.543
C08716=1019.870,153.547,382.289,167.701,51.319,159.542
C08717=1019.875,153.796,382.269,167.704,51.312,159.541
C08718=1019.880,154.045,382.248,167.708,51.305,159.540
C08719=1019.885,154.295,382.227,167.710,51.298,159.539
C08720=1019.891,154.544,382.207,167.715,51.290,159.538
C08721=1019.896,154.793,382.186,167.718,51.283,159.538
C08722=1019.902,155.075,382.162,167.722,51.275,159.536
C08723=1019.907,155.357,382.139,167.726,51.267,159.536
C08724=1019.914,155.639,382.116,167.730,51.259,159.535
C08725=1019.919,155.922,382.092,167.733,51.250,159.534
C08726=1019.925,156.170,382.071,167.736,51.243,159.533
C08727=1019.930,156.419,382.051,167.740,51.237,159.532
C08728=1019.935,156.669,382.029,167.744,51.229,159.531
C08729=1019.940,156.918,382.009,167.747,51.222,159.530
C08730=1019.945,157.167,381.988,167.750,51.214,159.529
C08731=1019.951,157.416,381.967,167.753,51.207,159.529
C08732=1019.956,157.665,381.947,167.758,51.200,159.528
C08733=1019.961,157.914,381.926,167.761,51.193,159.527
C08734=1019.967,158.163,381.905,167.764,51.186,159.526
C08735=1019.971,158.412,381.884,167.768,51.178,159.525
C08736=1019.977,158.661,381.863,167.771,51.171,159.524
C08737=1019.982,158.910,381.842,167.775,51.164,159.524
C08738=1019.987,159.160,381.821,167.778,51.157,159.523
C08739=1019.993,159.409,381.800,167.781,51.150,159.522
C08740=1019.997,159.658,381.779,167.785,51.142,159.521
C08741=1020.002,159.907,381.757,167.789,51.136,159.520
C08742=1020.007,160.156,381.736,167.792,51.129,159.520
C08743=1020.012,160.405,381.714,167.795,51.122,159.519
C08744=1020.017,160.654,381.694,167.799,51.115,159.518
C08745=1020.022,160.903,381.672,167.802,51.108,159.517
C08746=1020.027,161.152,381.651,167.806,51.101,159.517
C08747=1020.032,161.401,381.629,167.809,51.093,159.516
C08748=1020.037,161.650,381.608,167.813,51.086,159.515
C08749=1020.042,161.899,381.587,167.816,51.080,159.514
C08750=1020.047,162.148,381.566,167.820,51.073,159.513
C08751=1020.052,162.397,381.544,167.823,51.066,159.512
C08752=1020.057,162.645,381.523,167.827,51.059,159.512
C08753=1020.062,162.895,381.502,167.830,51.051,159.511
C08754=1020.067,163.144,381.479,167.834,51.044,159.510
C08755=1020.072,163.393,381.459,167.837,51.037,159.509
C08756=1020.077,163.642,381.437,167.841,51.030,159.509
C08757=1020.082,163.891,381.416,167.845,51.023,159.508
C08758=1020.087,164.140,381.395,167.848,51.017,159.507
C08759=1020.092,164.389,381.373,167.851,51.009,159.506
C08760=1020.097,164.638,381.352,167.855,51.002,159.505
C08761=1020.102,164.887,381.330,167.859,50.995,159.504
C08762=1020.108,165.136,381.309,167.862,50.988,159.504
C08763=1020.113,165.386,381.287,167.866,50.981,159.503
C08764=1020.118,165.634,381.266,167.870,50.974,159.502
C08765=1020.123,165.883,381.244,167.873,50.967,159.501
C08766=1020.128,166.132,381.223,167.876,50.960,159.500
C08767=1020.133,166.381,381.201,167.880,50.953,159.500
C08768=1020.139,166.630,381.180,167.884,50.946,159.499
C08769=1020.143,166.880,381.159,167.887,50.939,159.498
C08770=1020.148,167.129,381.137,167.890,50.931,159.497
C08771=1020.154,167.377,381.115,167.894,50.925,159.496
C08772=1020.158,167.626,381.094,167.898,50.917,159.496
C08773=1020.164,167.876,381.073,167.902,50.911,159.495
C08774=1020.169,168.125,381.051,167.905,50.904,159.494
C08775=1020.174,168.373,381.029,167.909,50.896,159.493
C08776=1020.179,168.622,381.008,167.912,50.889,159.492
C08777=1020.185,168.872,380.986,167.916,50.882,159.492
C08778=1020.189,169.121,380.964,167.920,50.875,159.491
C08779=1020.195,169.369,380.943,167.924,50.868,159.490
C08780=1020.200,169.618,380.921,167.927,50.861,159.489
C08781=1020.205,169.868,380.900,167.931,50.854,159.489
C08782=1020.210,170.117,380.878,167.934,50.847,159.488
C08783=1020.215,170.366,380.856,167.938,50.840,159.487
C08784=1020.221,170.614,380.835,167.942,50.833,159.486
C08785=1020.226,170.864,380.813,167.945,50.825,159.485
C08786=1020.232,171.146,380.789,167.949,50.817,159.484
C08787=1020.238,171.427,380.764,167.954,50.809,159.484
C08788=1020.243,171.709,380.740,167.958,50.801,159.483
C08789=1020.249,171.991,380.715,167.962,50.794,159.482
C08790=1020.256,172.240,380.693,167.966,50.787,159.481
C08791=1020.260,172.489,380.671,167.970,50.779,159.480
C08792=1020.265,172.738,380.650,167.973,50.772,159.479
C08793=1020.271,172.987,380.629,167.978,50.765,159.479
C08794=1020.276,173.236,380.607,167.981,50.758,159.478
C08795=1020.281,173.485,380.585,167.984,50.751,159.477
C08796=1020.287,173.734,380.563,167.988,50.744,159.476
C08797=1020.292,173.983,380.541,167.992,50.737,159.475
C08798=1020.297,174.232,380.520,167.996,50.730,159.475
C08799=1020.303,174.481,380.498,168.000,50.723,159.474
C08800=1020.308,174.730,380.476,168.003,50.716,159.473
C08801=1020.312,174.979,380.454,168.007,50.708,159.472
C08802=1020.319,175.228,380.433,168.011,50.701,159.471
C08803=1020.323,175.477,380.411,168.015,50.694,159.471
C08804=1020.329,175.726,380.389,168.018,50.688,159.470
C08805=1020.334,175.975,380.367,168.022,50.680,159.469
C08806=1020.339,176.224,380.345,168.026,50.673,159.468
C08807=1020.345,176.473,380.323,168.030,50.666,159.468
C08808=1020.350,176.722,380.302,168.034,50.659,159.467
C08809=1020.356,176.971,380.280,168.038,50.652,159.466
C08810=1020.360,177.220,380.258,168.041,50.644,159.465
C08811=1020.367,177.469,380.236,168.046,50.637,159.464
C08812=1020.371,177.718,380.214,168.049,50.631,159.464
C08813=1020.377,177.967,380.192,168.053,50.623,159.463
C08814=1020.382,178.216,380.171,168.057,50.617,159.462
C08815=1020.388,178.464,380.148,168.061,50.609,159.461
C08816=1020.393,178.714,380.126,168.064,50.602,159.460
C08817=1020.399,178.962,380.105,168.069,50.595,159.460
C08818=1020.404,179.212,380.082,168.072,50.588,159.459
C08819=1020.409,179.460,380.061,168.076,50.580,159.458
C08820=1020.415,179.710,380.039,168.080,50.574,159.457
C08821=1020.420,179.959,380.017,168.084,50.567,159.457
C08822=1020.425,180.207,379.994,168.088,50.560,159.456
C08823=1020.431,180.456,379.973,168.092,50.553,159.455
C08824=1020.436,180.705,379.951,168.095,50.545,159.454
C08825=1020.442,180.955,379.928,168.100,50.538,159.453
C08826=1020.447,181.203,379.907,168.103,50.531,159.453
C08827=1020.453,181.452,379.884,168.108,50.524,159.452
C08828=1020.458,181.701,379.862,168.112,50.517,159.451
C08829=1020.464,181.950,379.841,168.115,50.510,159.450
C08830=1020.469,182.199,379.819,168.119,50.503,159.450
C08831=1020.474,182.448,379.795,168.123,50.496,159.449
C08832=1020.479,182.698,379.773,168.126,50.489,159.448
C08833=1020.485,182.946,379.751,168.131,50.483,159.448
C08834=1020.489,183.196,379.728,168.135,50.476,159.447
C08835=1020.494,183.444,379.705,168.139,50.469,159.446
C08836=1020.500,183.694,379.683,168.143,50.462,159.445
C08837=1020.505,183.942,379.660,168.147,50.455,159.445
C08838=1020.510,184.192,379.637,168.150,50.448,159.444
C08839=1020.515,184.440,379.615,168.154,50.441,159.443
C08840=1020.520,184.689,379.592,168.158,50.434,159.442
C08841=1020.525,184.938,379.570,168.162,50.428,159.441
C08842=1020.530,185.187,379.547,168.167,50.421,159.441
C08843=1020.535,185.435,379.524,168.170,50.414,159.440
C08844=1020.540,185.685,379.501,168.175,50.407,159.440
C08845=1020.546,185.934,379.478,168.178,50.401,159.439
C08846=1020.551,186.182,379.456,168.183,50.394,159.438
C08847=1020.556,186.432,379.433,168.186,50.387,159.437
C08848=1020.561,186.680,379.410,168.191,50.380,159.437
C08849=1020.567,186.929,379.387,168.194,50.373,159.436
C08850=1020.572,187.210,379.362,168.198,50.366,159.435
C08851=1020.578,187.492,379.336,168.204,50.358,159.434
C08852=1020.584,187.773,379.310,168.208,50.350,159.433
C08853=1020.589,188.055,379.284,168.212,50.342,159.432
C08854=1020.595,188.304,379.261,168.216,50.335,159.432
C08855=1020.600,188.552,379.239,168.220,50.329,159.431
C08856=1020.605,188.802,379.216,168.225,50.322,159.430
C08857=1020.611,189.051,379.193,168.229,50.315,159.430
C08858=1020.616,189.299,379.170,168.233,50.308,159.429
C08859=1020.621,189.548,379.147,168.237,50.301,159.428
C08860=1020.626,189.797,379.124,168.241,50.295,159.428
C08861=1020.631,190.046,379.102,168.245,50.288,159.427
C08862=1020.636,190.295,379.079,168.248,50.281,159.426
C08863=1020.642,190.544,379.056,168.253,50.274,159.425
C08864=1020.647,190.792,379.033,168.257,50.268,159.425
C08865=1020.653,191.041,379.010,168.261,50.261,159.424
C08866=1020.658,191.290,378.987,168.266,50.254,159.423
C08867=1020.663,191.540,378.964,168.269,50.247,159.423
C08868=1020.668,191.788,378.942,168.274,50.240,159.422
C08869=1020.673,192.037,378.918,168.277,50.233,159.421
C08870=1020.679,192.286,378.895,168.282,50.226,159.420
C08871=1020.685,192.535,378.872,168.285,50.219,159.420
C08872=1020.689,192.784,378.849,168.290,50.213,159.419
C08873=1020.695,193.032,378.826,168.295,50.206,159.418
C08874=1020.701,193.281,378.803,168.298,50.199,159.418
C08875=1020.706,193.531,378.780,168.303,50.192,159.417
C08876=1020.711,193.779,378.757,168.307,50.185,159.416
C08877=1020.716,194.028,378.734,168.311,50.179,159.415
C08878=1020.722,194.277,378.711,168.315,50.172,159.415
C08879=1020.727,194.526,378.688,168.319,50.166,159.414
C08880=1020.732,194.775,378.664,168.324,50.159,159.413
C08881=1020.737,195.023,378.642,168.328,50.151,159.413
C08882=1020.743,195.272,378.619,168.332,50.145,159.412
C08883=1020.748,195.521,378.595,168.336,50.138,159.411
C08884=1020.754,195.770,378.572,168.341,50.131,159.410
C08885=1020.760,196.019,378.549,168.344,50.124,159.410
C08886=1020.765,196.268,378.526,168.349,50.118,159.409
C08887=1020.770,196.517,378.503,168.353,50.111,159.408
C08888=1020.775,196.765,378.480,168.357,50.104,159.408
C08889=1020.780,197.015,378.457,168.361,50.097,159.407
C08890=1020.786,197.263,378.434,168.366,50.090,159.406
C08891=1020.792,197.512,378.411,168.370,50.083,159.406
C08892=1020.797,197.761,378.386,168.374,50.077,159.405
C08893=1020.803,198.010,378.363,168.379,50.070,159.404
C08894=1020.809,198.259,378.341,168.383,50.063,159.404
C08895=1020.814,198.508,378.317,168.387,50.056,159.403
C08896=1020.819,198.757,378.294,168.391,50.049,159.402
C08897=1020.824,199.006,378.270,168.396,50.042,159.401
C08898=1020.830,199.255,378.248,168.401,50.036,159.401
C08899=1020.836,199.503,378.224,168.404,50.029,159.400
C08900=1020.841,199.752,378.201,168.409,50.022,159.399
C08901=1020.846,200.001,378.177,168.413,50.015,159.399
C08902=1020.852,200.249,378.154,168.417,50.009,159.398
C08903=1020.857,200.498,378.130,168.422,50.002,159.397
C08904=1020.862,200.747,378.106,168.427,49.996,159.397
C08905=1020.868,200.996,378.083,168.430,49.989,159.396
C08906=1020.873,201.245,378.059,168.435,49.982,159.395
C08907=1020.878,201.494,378.035,168.440,49.976,159.395
C08908=1020.883,201.743,378.011,168.443,49.969,159.394
C08909=1020.889,201.991,377.988,168.448,49.962,159.393
C08910=1020.894,202.240,377.964,168.453,49.956,159.393
C08911=1020.899,202.489,377.940,168.457,49.949,159.392
C08912=1020.904,202.738,377.916,168.461,49.943,159.391
C08913=1020.910,202.986,377.893,168.466,49.936,159.391
C08914=1020.932,204.025,377.793,168.907,50.030,159.483
C08915=1020.937,204.242,377.772,168.911,50.026,159.483
C08916=1020.943,204.459,377.749,168.914,50.021,159.482
C08917=1020.949,204.676,377.728,168.917,50.016,159.482
C08918=1020.954,204.892,377.706,168.920,50.011,159.481
C08919=1020.960,205.109,377.684,168.923,50.006,159.480
C08920=1020.966,205.326,377.662,168.927,50.001,159.480
C08921=1020.970,205.542,377.640,168.930,49.996,159.479
C08922=1020.976,205.760,377.617,168.933,49.991,159.479
C08923=1020.982,206.008,377.592,168.936,49.985,159.478
C08924=1020.988,206.256,377.566,168.940,49.980,159.478
C08925=1020.995,206.505,377.541,168.943,49.974,159.477
C08926=1021.001,206.754,377.515,168.947,49.968,159.476
C08927=1021.007,207.002,377.490,168.950,49.962,159.476
C08928=1021.013,207.251,377.465,168.954,49.957,159.475
C08929=1021.019,207.500,377.439,168.958,49.951,159.474
C08930=1021.026,207.748,377.414,168.961,49.946,159.474
C08931=1021.032,207.997,377.389,168.965,49.940,159.473
C08932=1021.038,208.245,377.363,168.968,49.935,159.473
C08933=1021.045,208.494,377.337,168.972,49.929,159.472
C08934=1021.050,208.743,377.311,168.975,49.924,159.471
C08935=1021.056,208.991,377.286,168.979,49.918,159.471
C08936=1021.063,209.239,377.260,168.982,49.913,159.470
C08937=1021.069,209.488,377.235,168.986,49.907,159.470
C08938=1021.076,209.738,377.209,168.989,49.902,159.469
C08939=1021.082,209.986,377.184,168.993,49.896,159.468
C08940=1021.088,210.234,377.158,168.996,49.891,159.468
C08941=1021.094,210.483,377.132,169.000,49.886,159.467
C08942=1021.100,210.732,377.106,169.003,49.880,159.467
C08943=1021.107,210.980,377.080,169.007,49.875,159.466
C08944=1021.112,211.229,377.054,169.010,49.869,159.465
C08945=1021.118,211.478,377.029,169.014,49.864,159.465
C08946=1021.125,211.726,377.003,169.017,49.858,159.464
C08947=1021.130,211.975,376.977,169.021,49.853,159.464
C08948=1021.137,212.223,376.951,169.024,49.848,159.463
C08949=1021.143,212.471,376.926,169.028,49.842,159.463
C08950=1021.149,212.721,376.899,169.032,49.837,159.462
C08951=1021.156,212.969,376.873,169.036,49.832,159.462
C08952=1021.162,213.218,376.848,169.039,49.826,159.461
C08953=1021.168,213.466,376.821,169.043,49.821,159.460
C08954=1021.174,213.715,376.796,169.046,49.816,159.460
C08955=1021.180,213.963,376.770,169.050,49.810,159.459
C08956=1021.186,214.212,376.744,169.053,49.805,159.459
C08957=1021.193,214.461,376.717,169.057,49.800,159.458
C08958=1021.199,214.709,376.692,169.060,49.794,159.457
C08959=1021.206,214.957,376.666,169.064,49.789,159.457
C08960=1021.211,215.206,376.640,169.068,49.784,159.457
C08961=1021.218,215.454,376.614,169.072,49.778,159.456
C08962=1021.224,215.704,376.588,169.075,49.773,159.455
C08963=1021.230,215.952,376.562,169.079,49.768,159.455
C08964=1021.236,216.201,376.536,169.082,49.763,159.454
C08965=1021.243,216.449,376.510,169.086,49.757,159.454
C08966=1021.248,216.698,376.484,169.089,49.752,159.453
C08967=1021.255,216.946,376.458,169.094,49.747,159.453
C08968=1021.262,217.194,376.432,169.097,49.742,159.452
C08969=1021.267,217.443,376.406,169.101,49.736,159.451
C08970=1021.274,217.692,376.380,169.104,49.731,159.451
C08971=1021.281,217.941,376.354,169.108,49.726,159.450
C08972=1021.287,218.189,376.328,169.111,49.721,159.450
C08973=1021.293,218.437,376.302,169.116,49.715,159.450
C08974=1021.299,218.686,376.275,169.119,49.711,159.449
C08975=1021.304,218.905,376.252,169.122,49.706,159.448
C08976=1021.310,219.125,376.229,169.126,49.701,159.448
C08977=1021.315,219.343,376.206,169.128,49.697,159.447
C08978=1021.321,219.562,376.182,169.132,49.692,159.447
C08979=1021.326,219.782,376.159,169.135,49.687,159.447
C08980=1021.332,220.001,376.136,169.138,49.683,159.446
C08981=1021.337,220.221,376.112,169.141,49.679,159.446
C08982=1021.342,220.439,376.089,169.144,49.674,159.445
C08983=1021.349,220.688,376.063,169.148,49.669,159.445
C08984=1021.355,220.937,376.037,169.152,49.664,159.444
C08985=1021.361,221.185,376.010,169.155,49.659,159.444
C08986=1021.367,221.433,375.984,169.159,49.654,159.443
C08987=1021.373,221.682,375.957,169.162,49.649,159.443
C08988=1021.379,221.931,375.930,169.167,49.644,159.442
C08989=1021.386,222.179,375.904,169.170,49.640,159.442
C08990=1021.392,222.428,375.877,169.173,49.635,159.441
C08991=1021.399,222.676,375.851,169.178,49.629,159.441
C08992=1021.404,222.925,375.825,169.181,49.624,159.440
C08993=1021.410,223.174,375.798,169.185,49.619,159.440
C08994=1021.417,223.422,375.772,169.188,49.614,159.439
C08995=1021.423,223.670,375.746,169.193,49.609,159.439
C08996=1021.429,223.919,375.719,169.196,49.604,159.438
C08997=1021.436,224.167,375.693,169.199,49.599,159.438
C08998=1021.442,224.416,375.666,169.204,49.595,159.438
C08999=1021.448,224.665,375.639,169.207,49.590,159.437
C09000=1021.454,224.913,375.613,169.211,49.584,159.437
C09001=1021.461,225.162,375.586,169.215,49.580,159.436
C09002=1021.467,225.410,375.560,169.218,49.575,159.435
C09003=1021.473,225.658,375.533,169.222,49.569,159.435
C09004=1021.479,225.907,375.506,169.226,49.565,159.435
C09005=1021.486,226.155,375.480,169.230,49.560,159.434
C09006=1021.492,226.404,375.453,169.233,49.555,159.434
C09007=1021.498,226.653,375.426,169.236,49.550,159.433
C09008=1021.505,226.901,375.400,169.241,49.545,159.433
C09009=1021.511,227.149,375.373,169.244,49.541,159.432
C09010=1021.517,227.398,375.346,169.249,49.535,159.432
C09011=1021.523,227.647,375.319,169.252,49.530,159.431
C09012=1021.529,227.895,375.292,169.255,49.526,159.431
C09013=1021.535,228.144,375.265,169.260,49.521,159.430
C09014=1021.542,228.392,375.238,169.263,49.516,159.430
C09015=1021.548,228.640,375.212,169.267,49.512,159.430
C09016=1021.554,228.889,375.185,169.271,49.507,159.429
C09017=1021.560,229.137,375.158,169.274,49.502,159.429
C09018=1021.567,229.386,375.131,169.278,49.497,159.428
C09019=1021.573,229.634,375.104,169.282,49.492,159.428
C09020=1021.579,229.883,375.077,169.286,49.488,159.427
C09021=1021.585,230.131,375.050,169.290,49.483,159.427
C09022=1021.592,230.380,375.023,169.293,49.479,159.427
C09023=1021.597,230.628,374.996,169.297,49.474,159.426
C09024=1021.604,230.877,374.968,169.301,49.469,159.426
C09025=1021.610,231.125,374.941,169.305,49.464,159.425
C09026=1021.616,231.374,374.914,169.308,49.460,159.425
C09027=1021.622,231.622,374.887,169.311,49.455,159.424
C09028=1021.629,231.871,374.860,169.316,49.451,159.424
C09029=1021.635,232.119,374.833,169.320,49.446,159.424
C09030=1021.641,232.368,374.806,169.323,49.441,159.423
C09031=1021.647,232.616,374.778,169.328,49.437,159.423
C09032=1021.653,232.865,374.751,169.331,49.432,159.422
C09033=1021.660,233.112,374.724,169.334,49.428,159.422
C09034=1021.666,233.361,374.697,169.339,49.423,159.422
C09035=1021.671,233.576,374.673,169.342,49.419,159.421
C09036=1021.677,233.792,374.650,169.345,49.415,159.421
C09037=1021.682,234.007,374.626,169.349,49.411,159.421
C09038=1021.687,234.222,374.603,169.351,49.407,159.420
C09039=1021.693,234.437,374.579,169.355,49.403,159.420
C09040=1021.698,234.652,374.556,169.358,49.399,159.420
C09041=1021.704,234.867,374.532,169.362,49.395,159.419
C09042=1021.709,235.083,374.508,169.365,49.391,159.419
C09043=1021.715,235.330,374.481,169.369,49.387,159.419
C09044=1021.722,235.579,374.453,169.373,49.382,159.418
C09045=1021.728,235.828,374.426,169.377,49.377,159.418
C09046=1021.734,236.076,374.399,169.380,49.373,159.417
C09047=1021.740,236.325,374.372,169.384,49.369,159.417
C09048=1021.747,236.573,374.344,169.388,49.364,159.417
C09049=1021.753,236.821,374.317,169.392,49.359,159.416
C09050=1021.760,237.070,374.290,169.396,49.355,159.416
C09051=1021.765,237.318,374.262,169.400,49.351,159.416
C09052=1021.772,237.566,374.234,169.404,49.346,159.415
C09053=1021.778,237.816,374.207,169.407,49.342,159.415
C09054=1021.784,238.063,374.180,169.412,49.337,159.414
C09055=1021.791,238.312,374.152,169.415,49.333,159.414
C09056=1021.797,238.561,374.125,169.419,49.329,159.414
C09057=1021.803,238.809,374.098,169.423,49.323,159.413
C09058=1021.810,239.057,374.070,169.427,49.319,159.413
C09059=1021.816,239.306,374.042,169.431,49.315,159.412
C09060=1021.822,239.553,374.014,169.435,49.310,159.412
C09061=1021.828,239.803,373.987,169.439,49.306,159.412
C09062=1021.834,240.051,373.959,169.442,49.302,159.412
C09063=1021.840,240.299,373.931,169.446,49.298,159.411
C09064=1021.847,240.547,373.904,169.451,49.293,159.411
C09065=1021.853,240.796,373.875,169.454,49.289,159.411
C09066=1021.859,241.044,373.848,169.458,49.285,159.410
C09067=1021.865,241.293,373.820,169.462,49.281,159.410
C09068=1021.872,241.541,373.792,169.466,49.276,159.410
C09069=1021.878,241.790,373.764,169.470,49.272,159.409
C09070=1021.884,242.038,373.736,169.474,49.268,159.409
C09071=1021.890,242.286,373.709,169.478,49.263,159.409
C09072=1021.897,242.535,373.681,169.482,49.259,159.408
C09073=1021.903,242.783,373.653,169.485,49.255,159.408
C09074=1021.909,243.031,373.625,169.489,49.251,159.407
C09075=1021.915,243.280,373.597,169.494,49.246,159.407
C09076=1021.922,243.528,373.569,169.497,49.242,159.407
C09077=1021.927,243.776,373.541,169.501,49.238,159.407
C09078=1021.934,244.025,373.513,169.505,49.233,159.406
C09079=1021.940,244.273,373.485,169.510,49.230,159.406
C09080=1021.946,244.522,373.456,169.513,49.225,159.406
C09081=1021.952,244.769,373.429,169.517,49.221,159.405
C09082=1021.958,245.018,373.400,169.520,49.217,159.405
C09083=1021.964,245.267,373.372,169.524,49.213,159.405
C09084=1021.970,245.515,373.344,169.529,49.209,159.405
C09085=1021.976,245.763,373.316,169.533,49.205,159.404
C09086=1021.982,246.011,373.287,169.536,49.200,159.404
C09087=1021.989,246.260,373.260,169.540,49.197,159.404
C09088=1021.995,246.509,373.231,169.545,49.192,159.403
C09089=1022.001,246.757,373.202,169.549,49.188,159.403
C09090=1022.007,247.004,373.175,169.553,49.185,159.403
C09091=1022.013,247.253,373.147,169.556,49.180,159.403
C09092=1022.019,247.501,373.117,169.561,49.176,159.402
C09093=1022.026,247.750,373.090,169.565,49.172,159.402
C09094=1022.032,247.999,373.061,169.569,49.168,159.402
C09095=1022.037,248.210,373.037,169.572,49.165,159.401
C09096=1022.042,248.423,373.013,169.576,49.161,159.401
C09097=1022.048,248.634,372.989,169.579,49.158,159.401
C09098=1022.053,248.847,372.964,169.583,49.155,159.401
C09099=1022.058,249.058,372.940,169.585,49.151,159.400
C09100=1022.064,249.270,372.916,169.589,49.147,159.400
